// Busca tempo de ciclo instantâneo/corrente das tarefas
GetTaskInfo (psAppName, Task_Information.TI_MainTask.psTaskName, Task_Information.TI_MainTask.pstTaskInfo);
GetTaskInfo (psAppName, Task_Information.TI_Configuration.psTaskName, Task_Information.TI_Configuration.pstTaskInfo);
GetTaskInfo (psAppName, Task_Information.TI_MODBUS_Client_2.psTaskName, Task_Information.TI_MODBUS_Client_2.pstTaskInfo);
GetTaskInfo (psAppName, Task_Information.TI_MODBUS_Client_3.psTaskName, Task_Information.TI_MODBUS_Client_3.pstTaskInfo);
GetTaskInfo (psAppName, Task_Information.TI_MODBUS_Master_1.psTaskName, Task_Information.TI_MODBUS_Master_1.pstTaskInfo);
GetTaskInfo (psAppName, Task_Information.TI_MODBUS_Server_2.psTaskName, Task_Information.TI_MODBUS_Server_2.pstTaskInfo);
GetTaskInfo (psAppName, Task_Information.TI_MODBUS_Server_3.psTaskName, Task_Information.TI_MODBUS_Server_3.pstTaskInfo);
GetTaskInfo (psAppName, Task_Information.TI_MODBUS_Slave_1.psTaskName, Task_Information.TI_MODBUS_Slave_1.pstTaskInfo);


// Se este for o PLCA e ele está no estado ativo...
IF DG_NX4010.tRedundancy.RedDgnLoc.sGeneral_Diag.ePLC_ID = CLUCONF_ID.PLC_A AND
   DG_NX4010.tRedundancy.RedDgnLoc.sGeneral_Diag.eRedState = REDUNDANCY_STATE.ACTIVE THEN
   
   	// Indica que existe um PLC ativo
	bPouActiveTime:= TRUE;
	
	// Atualiza variáveis de tempo de ciclo instantâneo/corrente das tarefas
	PersistentVars.dwPLCAMainTaskCurScanTime:= Task_Information.TI_MainTask.TaskInfo.dwCurScanTime;
	PersistentVars.dwPLCAConfigurationCurScanTime:= Task_Information.TI_Configuration.TaskInfo.dwCurScanTime;

	// Reseta variáveis de tempo de ciclo máximo e mínimo das tarefas caso solicitado
	IF Symbolics.bPlcAMaxMinSetup = TRUE THEN
		Symbolics.bPlcAMaxMinSetup:= FALSE;
		PersistentVars.dwPLCAMainTaskMaxScanTime:= PersistentVars.dwPLCAMainTaskCurScanTime;
		PersistentVars.dwPLCAMainTaskMinScanTime:= PersistentVars.dwPLCAMainTaskCurScanTime;
		PersistentVars.dwPLCAConfigurationMaxScanTime:= PersistentVars.dwPLCAConfigurationCurScanTime;
		PersistentVars.dwPLCAConfigurationMinScanTime:= PersistentVars.dwPLCAConfigurationCurScanTime;
	END_IF
	
	// Atualiza variáveis de tempo de ciclo máximo e mínimo das tarefas
	PersistentVars.dwPLCAMainTaskMaxScanTime:= MAX(PersistentVars.dwPLCAMainTaskMaxScanTime, PersistentVars.dwPLCAMainTaskCurScanTime);
	PersistentVars.dwPLCAMainTaskMinScanTime:= MIN(PersistentVars.dwPLCAMainTaskMinScanTime, PersistentVars.dwPLCAMainTaskCurScanTime);
	PersistentVars.dwPLCAConfigurationMaxScanTime:= MAX(PersistentVars.dwPLCAConfigurationMaxScanTime, PersistentVars.dwPLCAConfigurationCurScanTime);
	PersistentVars.dwPLCAConfigurationMinScanTime:= MIN(PersistentVars.dwPLCAConfigurationMinScanTime, PersistentVars.dwPLCAConfigurationCurScanTime);
	
	// Calcula tempo de ciclo médio da tarefa principal
	dwMainTaskSum:= dwMainTaskSum - adwAvgMainTask[iMainIndex];
	adwAvgMainTask[iMainIndex]:= PersistentVars.dwPLCAMainTaskCurScanTime;
	dwMainTaskSum:= dwMainTaskSum + adwAvgMainTask[iMainIndex];
	iMainIndex:= iMainIndex + 1;
	IF iMainIndex > DWORD_TO_INT(SIZEOF(adwAvgMainTask)/SIZEOF(adwAvgMainTask[1])) THEN
		iMainIndex:= 1;
	END_IF
	
	// Calcula tempo de ciclo médio da tarefa de configuração
	dwConfigTaskSum:= dwConfigTaskSum - adwAvgConfigTask[iConfigIndex];
	adwAvgConfigTask[iConfigIndex]:= PersistentVars.dwPLCAConfigurationCurScanTime;
	dwConfigTaskSum:= dwConfigTaskSum + adwAvgConfigTask[iConfigIndex];
	iConfigIndex:= iConfigIndex + 1;
	IF iConfigIndex > DWORD_TO_INT(SIZEOF(adwAvgConfigTask)/SIZEOF(adwAvgConfigTask[1])) THEN
		iConfigIndex:= 1;
	END_IF
	
	// Atualiza variáveis de tempo de ciclo médio das tarefas
	PersistentVars.dwPLCAMainTaskAvgScanTime:= dwMainTaskSum/(SIZEOF(adwAvgMainTask)/SIZEOF(adwAvgMainTask[1]));
	PersistentVars.dwPLCAConfigurationAvgScanTime:= dwConfigTaskSum/(SIZEOF(adwAvgConfigTask)/SIZEOF(adwAvgConfigTask[1]));

	// Registra percentual de uso da MainTask
	PersistentVars.dwPLCAMainTaskLoadMax:= MAX(PersistentVars.dwPLCAMainTaskLoadMax, (PersistentVars.dwPLCAMainTaskCurScanTime)/INT_TO_DWORD(ProjectConstants.iMainTaskInterval));
	PersistentVars.dwPLCAMainTaskLoadAvg:= (PersistentVars.dwPLCAMainTaskAvgScanTime)/INT_TO_DWORD(ProjectConstants.iMainTaskInterval);
	PersistentVars.dwPLCAMainTaskLoadMin:= MIN(PersistentVars.dwPLCAMainTaskLoadMin, (PersistentVars.dwPLCAMainTaskCurScanTime)/INT_TO_DWORD(ProjectConstants.iMainTaskInterval));
END_IF

// Se este for o PLCB e ele está no estado ativo...
IF DG_NX4010.tRedundancy.RedDgnLoc.sGeneral_Diag.ePLC_ID = CLUCONF_ID.PLC_B AND
   DG_NX4010.tRedundancy.RedDgnLoc.sGeneral_Diag.eRedState = REDUNDANCY_STATE.ACTIVE THEN
	
   	// Indica que existe um PLC ativo
	bPouActiveTime:= TRUE;
	
	// Atualiza variáveis de tempo de ciclo instantâneo/corrente das tarefas
	PersistentVars.dwPLCBMainTaskCurScanTime:= Task_Information.TI_MainTask.TaskInfo.dwCurScanTime;
	PersistentVars.dwPLCBConfigurationCurScanTime:= Task_Information.TI_Configuration.TaskInfo.dwCurScanTime;
	
	// Reseta variáveis de tempo de ciclo máximo e mínimo das tarefas caso solicitado
	IF Symbolics.bPlcBMaxMinSetup = TRUE THEN
		Symbolics.bPlcBMaxMinSetup:= FALSE;	
		PersistentVars.dwPLCBMainTaskMaxScanTime:= PersistentVars.dwPLCBMainTaskCurScanTime;
		PersistentVars.dwPLCBMainTaskMinScanTime:= PersistentVars.dwPLCBMainTaskCurScanTime;
		PersistentVars.dwPLCBConfigurationMaxScanTime:= PersistentVars.dwPLCBConfigurationCurScanTime;
		PersistentVars.dwPLCBConfigurationMinScanTime:= PersistentVars.dwPLCBConfigurationCurScanTime;
	END_IF
	
	// Atualiza variáveis de tempo de ciclo máximo e mínimo das tarefas
	PersistentVars.dwPLCBMainTaskMaxScanTime:= MAX(PersistentVars.dwPLCBMainTaskMaxScanTime, PersistentVars.dwPLCBMainTaskCurScanTime);
	PersistentVars.dwPLCBMainTaskMinScanTime:= MIN(PersistentVars.dwPLCBMainTaskMinScanTime, PersistentVars.dwPLCBMainTaskCurScanTime);
	PersistentVars.dwPLCBConfigurationMaxScanTime:= MAX(PersistentVars.dwPLCBConfigurationMaxScanTime, PersistentVars.dwPLCBConfigurationCurScanTime);
	PersistentVars.dwPLCBConfigurationMinScanTime:= MIN(PersistentVars.dwPLCBConfigurationMinScanTime, PersistentVars.dwPLCBConfigurationCurScanTime);
	
	// Calcula tempo de ciclo médio da tarefa principal
	dwMainTaskSum:= dwMainTaskSum - adwAvgMainTask[iMainIndex];
	adwAvgMainTask[iMainIndex]:= PersistentVars.dwPLCBMainTaskCurScanTime;
	dwMainTaskSum:= dwMainTaskSum + adwAvgMainTask[iMainIndex];
	iMainIndex:= iMainIndex + 1;
	IF iMainIndex > DWORD_TO_INT(SIZEOF(adwAvgMainTask)/SIZEOF(adwAvgMainTask[1])) THEN
		iMainIndex:= 1;
	END_IF
	
	// Calcula tempo de ciclo médio da tarefa de configuração
	dwConfigTaskSum:= dwConfigTaskSum - adwAvgConfigTask[iConfigIndex];
	adwAvgConfigTask[iConfigIndex]:= PersistentVars.dwPLCBConfigurationCurScanTime;
	dwConfigTaskSum:= dwConfigTaskSum + adwAvgConfigTask[iConfigIndex];
	iConfigIndex:= iConfigIndex + 1;
	IF iConfigIndex > DWORD_TO_INT(SIZEOF(adwAvgConfigTask)/SIZEOF(adwAvgConfigTask[1])) THEN
		iConfigIndex:= 1;
	END_IF
	
	// Atualiza variáveis de tempo de ciclo médio das tarefas
	PersistentVars.dwPLCBMainTaskAvgScanTime:= dwMainTaskSum/(SIZEOF(adwAvgMainTask)/SIZEOF(adwAvgMainTask[1]));
	PersistentVars.dwPLCBConfigurationAvgScanTime:= dwConfigTaskSum/(SIZEOF(adwAvgConfigTask)/SIZEOF(adwAvgConfigTask[1]));
	
	// Registra percentual de uso da MainTask
	PersistentVars.dwPLCBMainTaskLoadMax:= MAX(PersistentVars.dwPLCBMainTaskLoadMax, (PersistentVars.dwPLCBMainTaskCurScanTime)/INT_TO_DWORD(ProjectConstants.iMainTaskInterval));
	PersistentVars.dwPLCBMainTaskLoadAvg:= (PersistentVars.dwPLCBMainTaskAvgScanTime)/INT_TO_DWORD(ProjectConstants.iMainTaskInterval);
	PersistentVars.dwPLCBMainTaskLoadMin:= MIN(PersistentVars.dwPLCBMainTaskLoadMin, (PersistentVars.dwPLCBMainTaskCurScanTime)/INT_TO_DWORD(ProjectConstants.iMainTaskInterval));
END_IF

// Calcula o tempo mínimo total, somando a duração mínima de todas as POUs, menos da MainPrg
MinMaxTimes.uliPouMinTime_TOTAL:=	MinMaxTimes.uliPouMinTime_Alarms +
						MinMaxTimes.uliPouMinTime_CheckIec104 +
						MinMaxTimes.uliPouMinTime_CheckLanguages +
						MinMaxTimes.uliPouMinTime_CheckProfibusIOs +
						MinMaxTimes.uliPouMinTime_CheckRecipe +
						MinMaxTimes.uliPouMinTime_CheckSoe +
						MinMaxTimes.uliPouMinTime_IncrRedData +
						MinMaxTimes.uliPouMinTime_PidGenerator +
						MinMaxTimes.uliPouMinTime_StateChange +
						MinMaxTimes.uliPouMinTime_CheckDiags +
						MinMaxTimes.uliPouMinTime_CheckForcing +		
						MinMaxTimes.uliPouMinTime_CheckModbus1 +
						MinMaxTimes.uliPouMinTime_CheckModbus2 +
						MinMaxTimes.uliPouMinTime_CheckModbus3 +
						MinMaxTimes.uliPouMinTime_CheckModbus4 +
						MinMaxTimes.uliPouMinTime_CheckRam +
						MinMaxTimes.uliPouMinTime_CheckRedData +
						MinMaxTimes.uliPouMinTime_CheckSntp +
						MinMaxTimes.uliPouMinTime_CleanStatus +
						MinMaxTimes.uliPouMinTime_CycleTimes +
						//MinMaxTimes.uliPouMinTime_DaylightSavingTime +
						MinMaxTimes.uliPouMinTime_UserLog +
						MinMaxTimes.uliPouMinTime_WriteHwVersionsNonActive+
						MinMaxTimes.uliPouMinTime_CheckNVL +
						MinMaxTimes.uliPouMinTime_MQTT;
						
// Calcula o tempo máximo total, somando a duração máxima de todas as POUs, menos da MainPrg
MinMaxTimes.uliPouMaxTime_TOTAL:=	MinMaxTimes.uliPouMaxTime_Alarms +
						MinMaxTimes.uliPouMaxTime_CheckIec104 +
						MinMaxTimes.uliPouMaxTime_CheckLanguages +
						MinMaxTimes.uliPouMaxTime_CheckProfibusIOs + 
						MinMaxTimes.uliPouMaxTime_CheckRecipe +
						MinMaxTimes.uliPouMaxTime_CheckSoe +
						MinMaxTimes.uliPouMaxTime_IncrRedData +
						MinMaxTimes.uliPouMaxTime_PidGenerator +
						MinMaxTimes.uliPouMaxTime_StateChange +
						MinMaxTimes.uliPouMaxTime_CheckDiags +
						MinMaxTimes.uliPouMaxTime_CheckForcing +		
						MinMaxTimes.uliPouMaxTime_CheckModbus1 +
						MinMaxTimes.uliPouMaxTime_CheckModbus2 +
						MinMaxTimes.uliPouMaxTime_CheckModbus3 +
						MinMaxTimes.uliPouMaxTime_CheckModbus4 +
						MinMaxTimes.uliPouMaxTime_CheckRam +
						MinMaxTimes.uliPouMaxTime_CheckRedData +
						MinMaxTimes.uliPouMaxTime_CheckSntp +
						MinMaxTimes.uliPouMaxTime_CleanStatus +
						MinMaxTimes.uliPouMaxTime_CycleTimes +
						//MinMaxTimes.uliPouMaxTime_DaylightSavingTime +
						MinMaxTimes.uliPouMaxTime_UserLog +
						MinMaxTimes.uliPouMaxTime_WriteHwVersionsNonActive+
						MinMaxTimes.uliPouMaxTime_CheckNVL+
						MinMaxTimes.uliPouMaxTime_MQTT;

// Registra o tempo do sistema
SysTimeGetUs(uliPouEndTime);
// Calcula duração mínima/máxima desta POU, se um dos PLCs está ativo
IF bPouActiveTime THEN
	MinMaxTimes.uliPouMinTime_CycleTimes:= MIN(MinMaxTimes.uliPouMinTime_CycleTimes, uliPouEndTime - uliPouIniTime);
	MinMaxTimes.uliPouMaxTime_CycleTimes:= MAX(MinMaxTimes.uliPouMaxTime_CycleTimes, uliPouEndTime - uliPouIniTime);
END_IF

END_PROGRAM

// Device/Application/UserPOUs/Non-Redundant/CheckModbus1
PROGRAM CheckModbus1
VAR
	byIndex : BYTE;
	wIndex : WORD;
	bStatusCoil : BOOL;
	bStatusStatus : BOOL;
	bStatusHolding : BOOL;
	bStatusInputReg : BOOL;
	liDigitalTimer : LINT := 0;
	liAnalogTimer : LINT := 0;
	abyCoilsError_DataWr : ARRAY [0..119] OF BYTE;
	abyCoilsError_DataRd : ARRAY [0..119] OF BYTE;
	abyStatusError_DataWr : ARRAY [0..119] OF BYTE;
	abyStatusError_DataRd : ARRAY [0..119] OF BYTE;
	awHoldingError_DataWr : ARRAY [0..119] OF WORD;
	awHoldingError_DataRd : ARRAY [0..119] OF WORD;
	awInputRegError_DataWr : ARRAY [0..119] OF WORD;
	awInputRegError_DataRd : ARRAY [0..119] OF WORD;
	wOldRXNormalResponses : WORD;
	iMilisecondsCounter : INT;
	iBytesPerResponse : INT := 240;
	uliPouIniTime : ULINT;
	uliPouEndTime : ULINT;
END_VAR

// Consistencia da integridade dos dados trocados via MODBUS 1

// Registra o tempo do sistema
SysTimeGetUs(uliPouIniTime);

//
// Controle e consistência dos coils e input status
//

// Consiste os valores lidos
bStatusCoil:= TRUE;
bStatusStatus:= TRUE;
FOR byIndex:= 0 TO 119 BY 1 DO
	bStatusCoil:= bStatusCoil AND (ATs.abyModbus1CoilsRead[byIndex] = ATs.abyModbus1CoilsWrite[byIndex]);
	bStatusStatus:= bStatusStatus AND (ATs.abyModbus1StatusRead[byIndex] = ATs.abyModbus1CoilsWrite[byIndex]);
END_FOR

// Se o protocolo MODBUS está rodando e se os dados são consistentes...
IF DG_MODBUS_Master_1.tDiag.bRunning AND bStatusCoil AND bStatusStatus THEN
	// Altera o valor a ser escrito nos coils
	ATs.abyModbus1CoilsWrite[0]:= ATs.abyModbus1CoilsWrite[0] + 10;
	// Reseta o temporizador
	liDigitalTimer:= 0;
ELSE
	// Acumula o tempo que passou
	liDigitalTimer:= liDigitalTimer + ProjectConstants.iMainTaskInterval;
	// Registra o tempo máximo
	MinMaxTimes.liDigMaxTime_CheckModbus1:= MAX(MinMaxTimes.liDigMaxTime_CheckModbus1, liDigitalTimer);
	// Caso o tempo máximo tenha sido extrapolado...
	IF liDigitalTimer >= ProjectConstants.iModbus1ReadWriteDelay THEN
		// Registra falha nos coils, caso tenha ocorrido
		IF bStatusCoil = FALSE THEN
			NonRedPointer.pbModbus1ErrorCoilLoc^:= TRUE;
			abyCoilsError_DataWr:= ATs.abyModbus1CoilsWrite;
			abyCoilsError_DataRd:= ATs.abyModbus1CoilsRead;		
		END_IF
		// Registra falha nos inputs, caso tenha ocorrido
		IF bStatusStatus = FALSE THEN
			NonRedPointer.pbModbus1ErrorStatusLoc^:= TRUE;
			abyStatusError_DataWr:= ATs.abyModbus1CoilsWrite;
			abyStatusError_DataRd:= ATs.abyModbus1StatusRead;
		END_IF
	END_IF
END_IF

// Atualiza os valores escritos
FOR byIndex:= 1 TO 119 BY 1 DO
	ATs.abyModbus1CoilsWrite[byIndex]:= ATs.abyModbus1CoilsWrite[byIndex - 1] + byIndex;
END_FOR

//
// Controle e consistência dos holding e input registers
//

// Consiste os valores lidos
bStatusHolding:= TRUE;
bStatusInputReg:= TRUE;
FOR wIndex:= 0 TO 119 BY 1 DO
	bStatusHolding:= bStatusHolding AND (ATs.awModbus1HoldingRead[wIndex] = ATs.awModbus1HoldingWrite[wIndex]);
	bStatusInputReg:= bStatusInputReg AND (ATs.awModbus1InputRegRead[wIndex] = ATs.awModbus1HoldingWrite[wIndex]);
END_FOR

// Se o protocolo MODBUS está rodando e se os dados são consistentes...
IF DG_MODBUS_Master_1.tDiag.bRunning AND bStatusHolding AND bStatusInputReg THEN
	// Incrementa o valor escrito nos holding registers
	ATs.awModbus1HoldingWrite[0]:= ATs.awModbus1HoldingWrite[0] + 100;
	// Reseta o temporizador
	liAnalogTimer:= 0;
ELSE
	// Acumula o tempo que passou
	liAnalogTimer:= liAnalogTimer + ProjectConstants.iMainTaskInterval;
	// Registra o tempo máximo
	MinMaxTimes.liAnaMaxTime_CheckModbus1:= MAX(MinMaxTimes.liAnaMaxTime_CheckModbus1, liAnalogTimer);
	// Caso o tempo máximo tenha sido extrapolado...
	IF liAnalogTimer >= ProjectConstants.iModbus1ReadWriteDelay THEN
		// Registra falha nos holding register, caso tenha ocorrido
		IF bStatusHolding = FALSE THEN
			NonRedPointer.pbModbus1ErrorHoldingLoc^:= TRUE;
			awHoldingError_DataWr:= ATs.awModbus1HoldingWrite;
			awHoldingError_DataRd:= ATs.awModbus1HoldingRead;
		END_IF
		// Registra falha nos input register, caso tenha ocorrido
		IF bStatusInputReg = FALSE THEN
			NonRedPointer.pbModbus1ErrorInputRegLoc^:= TRUE;
			awInputRegError_DataWr:= ATs.awModbus1HoldingWrite;
			awInputRegError_DataRd:= ATs.awModbus1InputRegRead;
		END_IF
	END_IF
END_IF

// Atualiza os valores escritos
FOR wIndex:= 1 TO 119 BY 1 DO
	ATs.awModbus1HoldingWrite[wIndex]:= ATs.awModbus1HoldingWrite[wIndex - 1] + wIndex;
END_FOR

//
// Calcula a taxa média de comunicação
//

// Incrementa o número de milisegundos que transcorreram
iMilisecondsCounter:= iMilisecondsCounter + ProjectConstants.iMainTaskInterval;
// Se já se passou o tempo configurado desde a última média realizada...
IF iMilisecondsCounter >= ProjectConstants.iMsToComputeComRate THEN
	// Só calcula se o contador não virou
	IF DG_MODBUS_Master_1.tStat.wRXNormalResponses > wOldRXNormalResponses THEN
		// Calcula a taxa de comunicação atual
		MinMaxTimes.diModbus1BytesPerSec:=	WORD_TO_DINT(DG_MODBUS_Master_1.tStat.wRXNormalResponses - wOldRXNormalResponses) *
											iBytesPerResponse * 1000 / iMilisecondsCounter;
	END_IF
	// Zera o número de milisegundos transcorridos
	iMilisecondsCounter:= 0;
	// Salva número de respostas atuais
	wOldRXNormalResponses:= DG_MODBUS_Master_1.tStat.wRXNormalResponses;
END_IF

PersistentVars.bModbus1ErrorCoil:=		NonRedPointer.pbModbus1ErrorCoilLoc^ OR
										NonRedPointer.pbModbus1ErrorCoilRem^;
PersistentVars.bModbus1ErrorStatus:=	NonRedPointer.pbModbus1ErrorStatusLoc^ OR
										NonRedPointer.pbModbus1ErrorStatusRem^;
PersistentVars.bModbus1ErrorHolding:=	NonRedPointer.pbModbus1ErrorHoldingLoc^ OR
										NonRedPointer.pbModbus1ErrorHoldingRem^;
PersistentVars.bModbus1ErrorInputReg:=	NonRedPointer.pbModbus1ErrorInputRegLoc^ OR
										NonRedPointer.pbModbus1ErrorInputRegRem^;

// Registra o tempo do sistema
SysTimeGetUs(uliPouEndTime);
// Calcula duração mínima/máxima desta POU
MinMaxTimes.uliPouMinTime_CheckModbus1:= MIN(MinMaxTimes.uliPouMinTime_CheckModbus1, uliPouEndTime - uliPouIniTime);
MinMaxTimes.uliPouMaxTime_CheckModbus1:= MAX(MinMaxTimes.uliPouMaxTime_CheckModbus1, uliPouEndTime - uliPouIniTime);

END_PROGRAM

// Device/Application/UserPOUs/Redundant/ProfibusStateChange
PROGRAM ProfibusStateChange
VAR
	byState : BYTE := 1;
	iTime : INT := 0;
	iLimit : INT := ProjectConstants.iLowLimit;
	bLastState : BOOL;
	uliPouIniTime : ULINT;
	uliPouEndTime : ULINT;
END_VAR

 // Esta POU alterna o estado de redundância das remotas Profibus automaticamente.
// Ela é chamada pela POU CheckProfibusIOs, portanto ela é executada somente pelo CP ativo,
// isto deve ser levado em consideração para compreender o código abaixo.
// Estado inicial: Remota A ativo, Remota B stand-by.

// Registra o tempo do sistema
SysTimeGetUs(uliPouIniTime);

CASE byState OF
	
	1:	// Aguarda tempo para estabilização da nova remota ativa
		IF iTime < ProjectConstants.iTimeToSkipAsActive THEN
			iTime:= iTime + ProjectConstants.iMainTaskInterval;
		ELSE
			// Próximo estado
			byState:= 2;
			// Joga zero para os bits de switch over das remotas ponto para que estas o executem
			REM05_PO5065_OUT:= 0;
			REM10_PO5065_OUT:= 0;
		END_IF
	
	2:	// Aguarda iLimit ciclos para a próxima alteração de estados
		IF iTime < iLimit THEN
			iTime:= iTime + ProjectConstants.iMainTaskInterval;
		ELSE
			byState:= 3;
		END_IF
	
	3:	// Realiza switchover
		PersistentVars.dwPBSwitchoverCnt:= PersistentVars.dwPBSwitchoverCnt + 1;
		IF bLastState THEN
			REM05_PO5065_OUT:= 1024;
			REM10_PO5065_OUT:= 1024;
			bLastState:=FALSE;
		ELSE
			REM05_PO5065_OUT:= 768;
			REM10_PO5065_OUT:= 768;
			bLastState:=TRUE;
		END_IF			
		byState:= 4;
		iTime:= 0;
			
	4: 	// Incrementa o valor limite para troca de estados
		iLimit:= iLimit + ProjectConstants.iMainTaskInterval;
		// Mantém a duração de cada estado entre 50 e 250 ciclos
		IF iLimit > ProjectConstants.iHighLimit THEN
			iLimit:= ProjectConstants.iLowLimit;
		END_IF
		// Inicia um novo ciclo de troca de estados
		byState:= 1;
END_CASE

// Registra o tempo do sistema
SysTimeGetUs(uliPouEndTime);
// Calcula duração mínima/máxima desta POU
MinMaxTimes.uliPouMinTime_ProfibusStateChange:= MIN(MinMaxTimes.uliPouMinTime_ProfibusStateChange, uliPouEndTime - uliPouIniTime);
MinMaxTimes.uliPouMaxTime_ProfibusStateChange:= MAX(MinMaxTimes.uliPouMaxTime_ProfibusStateChange, uliPouEndTime - uliPouIniTime);

END_PROGRAM

// Device/Application/UserPOUs/Non-Redundant/CheckRam
PROGRAM CheckRam
VAR
	stRamInfo : SYSTEM_RAM_INFO_T;
	dwRamTotalError : DWORD;
	dwRamFreeError : DWORD;
	uliPouIniTime : ULINT;
	uliPouEndTime : ULINT;
	bInternalFlag : BOOL;
END_VAR

// POU para consistência da memória RAM total e livre.

// Registra o tempo do sistema
SysTimeGetUs(uliPouIniTime);

// Busca as informações da memória RAM apenas no primeiro ciclo como inativo, pois a função consome muito tempo
IF DG_NX4010.tRedundancy.RedDgnLoc.sGeneral_Diag.eRedState = REDUNDANCY_STATE.INACTIVE  AND NonRedData.bRedStateChanged  THEN
	// Atualiza as informações a respeito da memória RAM
	SystemRamInfoGet(stRamInfo);
	// Flag para indicar se passou pelo estado inativo para habiltiar a consistencia do teste na inicialização do teste
	IF stRamInfo.dwTotal > 0 AND stRamInfo.dwFree > 0 THEN
		bInternalFlag:= TRUE;
	END_IF
END_IF

// Consiste a memória RAM apenas no primeiro ciclo como ativo (a UCP não ativa não consegue escrever nas PersistentVars)  
IF 	DG_NX4010.tRedundancy.RedDgnLoc.sGeneral_Diag.eRedState = REDUNDANCY_STATE.ACTIVE AND NonRedData.bRedStateChanged AND bInternalFlag THEN

		// Consistência da memória RAM total
		IF stRamInfo.dwTotal <> ProjectConstants.dwRamTotal THEN
			dwRamTotalError:= stRamInfo.dwTotal;
			NonRedPointer.pbRamTotalFailureLoc^:= TRUE;
		END_IF
	// Registra os valores mínimos e máximos e consiste a variação de memória livre
			IF DG_NX4010.tRedundancy.RedDgnLoc.sGeneral_Diag.ePLC_ID = CLUCONF_ID.PLC_A THEN
				// Registra valores de memória RAM livre mínima e máxima do PLC correspondente
				PersistentVars.dwMinFreeRamPlcA:= MIN(PersistentVars.dwMinFreeRamPlcA, stRamInfo.dwFree/1024);
				PersistentVars.dwMaxFreeRamPlcA:= MAX(PersistentVars.dwMaxFreeRamPlcA, stRamInfo.dwFree/1024);
				PersistentVars.dwInstFreeRamPlcA:= stRamInfo.dwFree/1024;
				// Consistência da variação da memória RAM livre
				IF PersistentVars.dwMaxFreeRamPlcA - PersistentVars.dwMinFreeRamPlcA > ProjectConstants.dwRamVariance THEN
					dwRamFreeError:= PersistentVars.dwMaxFreeRamPlcA;
					NonRedPointer.pbRamFreeVarFailureLoc^:= TRUE;
				END_IF
			ELSE
				// Registra valores de memória RAM livre mínima e máxima do PLC correspondente
				PersistentVars.dwMinFreeRamPlcB:= MIN(PersistentVars.dwMinFreeRamPlcB, stRamInfo.dwFree/1024);
				PersistentVars.dwMaxFreeRamPlcB:= MAX(PersistentVars.dwMaxFreeRamPlcB, stRamInfo.dwFree/1024);
				PersistentVars.dwInstFreeRamPlcB:= stRamInfo.dwFree/1024;
				// Consistência da variação da memória RAM livre
				IF PersistentVars.dwMaxFreeRamPlcB - PersistentVars.dwMinFreeRamPlcB > ProjectConstants.dwRamVariance THEN
					dwRamFreeError:= PersistentVars.dwMaxFreeRamPlcB;
					NonRedPointer.pbRamFreeVarFailureLoc^:= TRUE;
				END_IF
			END_IF
	// Reinicializa flag de teste
	bInternalFlag:= FALSE;
END_IF

// Inicializa os diagnósticos locais/remotos se solicitado
IF SymbolicsNonRedundant.bEnableCleanStats_CheckRam THEN
	NonRedPointer.pbRamTotalFailureLoc^:= FALSE;
	NonRedPointer.pbRamFreeVarFailureLoc^:= FALSE;
	NonRedPointer.pbRamTotalFailureRem^:= FALSE;
	NonRedPointer.pbRamFreeVarFailureRem^:= FALSE;	
	// Reinicializa flag de teste
	bInternalFlag:= FALSE;
	// Inicializa os valores atualizados pela função SystemRamInfoGet
	stRamInfo.dwTotal:= 0;
	stRamInfo.dwFree:= 0;
	SymbolicsNonRedundant.bEnableCleanStats_CheckRam := FALSE;
END_IF

// Atribui as variáveis locais/remotas de falha às variáveis redundantes persistentes

PersistentVars.bRamTotalFailure:=	PersistentVars.bRamTotalFailure OR
									NonRedPointer.pbRamTotalFailureLoc^ OR
									NonRedPointer.pbRamTotalFailureRem^;
PersistentVars.bRamFreeVarFailure:=	PersistentVars.bRamFreeVarFailure OR
									NonRedPointer.pbRamFreeVarFailureLoc^ OR
									NonRedPointer.pbRamFreeVarFailureRem^;

// Registra o tempo do sistema
SysTimeGetUs(uliPouEndTime);
// Calcula duração mínima/máxima desta POU
MinMaxTimes.uliPouMinTime_CheckRam:= MIN(MinMaxTimes.uliPouMinTime_CheckRam, uliPouEndTime - uliPouIniTime);
MinMaxTimes.uliPouMaxTime_CheckRam:= MAX(MinMaxTimes.uliPouMaxTime_CheckRam, uliPouEndTime - uliPouIniTime);

END_PROGRAM

// Device/Application/UserPOUs/Non-Redundant/CheckSntp
PROGRAM CheckSntp
VAR CONSTANT
	byDelay : BYTE := 10;
	iSntpTolerance : INT := (21200); // = 20000 + 1200
END_VAR
VAR
	sCurrentTime : NextoStandard.EXTENDED_DATE_AND_TIME;
	sGetTime : NextoStandard.EXTENDED_DATE_AND_TIME;
	sSetTime : NextoStandard.SetDateAndTime;
	GetTimeZone_Status : RTC_STATUS;
	TimeZone : TIMEZONESETTINGS;
	bStartup : BOOL := TRUE;
	byState : BYTE := 1;
	bSignal : BOOL := FALSE;
	iSyncCounter : INT := 0;
	dwReference : DWORD := 0;
	liSntpMsTimer : LINT := 0;
	uliPouIniTime : ULINT;
	uliPouEndTime : ULINT;
END_VAR

// Teste que verifica a atualização do relógio pelo SNTP
// SETUP: Configurar o SNTP para 20s de period, com 150ms de minimum error

// Registra o tempo do sistema
SysTimeGetUs(uliPouIniTime);

// Testa se a função GetTimeZone estrá retornando os valores corretos
GetTimeZone_Status := GetTimeZone(TimeZone);
IF GetTimeZone_Status <> RTC_STATUS.NO_ERROR OR TimeZone.iHour <> -3 OR TimeZone.iMinutes <> 0 THEN
	PersistentVars.bTimezoneFailure := TRUE;
END_IF

// Acumula o tempo que passou
liSntpMsTimer:= liSntpMsTimer + ProjectConstants.iMainTaskInterval;

// Verifica se o serviço está funcionando
IF	DG_NX3030.tDetailed.SNTP.bServiceEnabled = TRUE AND
	DG_NX3030.tDetailed.SNTP.byActiveTimeServer <> NO_TIME_SERVER THEN
		// Correção inicial da referência
		IF bStartup = TRUE THEN
			// Correção inicial da referência
			dwReference:= DG_NX3030.tDetailed.SNTP.dwRTCTimeUpdatedCount;
			// Restaura variáveis locais não retentivas
			NonRedPointer.pbSntpServerFailuresLoc^:= PersistentVars.bSntpServerFailures;
			NonRedPointer.pbSntpSourceFailuresLoc^:= PersistentVars.bSntpSourceFailures;
			NonRedPointer.piSntpSyncFailuresLoc^:= PersistentVars.iSntpSyncFailures;
			// Reseta indicação de inicialização
			bStartup:= FALSE;
		END_IF
		
		CASE byState OF
			
			1:	// Armazena o horário atual em sCurrentTime, confere se a atualização anterior ocorreu
				NextoStandard.GetDateAndTime(sGetTime);
				sCurrentTime.byDayOfMonth:= sGetTime.byDayOfMonth;
				sCurrentTime.byHours:= sGetTime.byHours;
				sCurrentTime.byMinutes:= sGetTime.byMinutes;
				sCurrentTime.byMonth:= sGetTime.byMonth;
				sCurrentTime.bySeconds:= sGetTime.bySeconds;
				sCurrentTime.wMilliseconds:= sGetTime.wMilliseconds;
				sCurrentTime.wYear:= sGetTime.wYear;
				// Se o contador está diferente da referência, indica erro na sincronização
				IF DG_NX3030.tDetailed.SNTP.dwRTCTimeUpdatedCount < dwReference THEN
					IF NonRedPointer.piSntpSyncFailuresLoc^ < ProjectConstants.iValueRedLimit THEN
						NonRedPointer.piSntpSyncFailuresLoc^:= NonRedPointer.piSntpSyncFailuresLoc^+1;
					END_IF
					dwReference:= DG_NX3030.tDetailed.SNTP.dwRTCTimeUpdatedCount;
				// Indica que houve 2 atualizações no intervalo, o que não pode ser considerado uma falha
				ELSIF DG_NX3030.tDetailed.SNTP.dwRTCTimeUpdatedCount > dwReference THEN
					dwReference:= DG_NX3030.tDetailed.SNTP.dwRTCTimeUpdatedCount;
				END_IF				
				byState:= 2;
			
			2:	// Adianta ou atrasa sCurrentTime em 10s alternadamente
				IF bSignal = TRUE THEN
					IF sCurrentTime.bySeconds >= byDelay THEN
						sCurrentTime.bySeconds:= sCurrentTime.bySeconds - byDelay;
						byState:= 3;
					ELSE
						byState:= 1;
					END_IF
				ELSE
					IF sCurrentTime.bySeconds < (60 - byDelay) THEN
						sCurrentTime.bySeconds:= sCurrentTime.bySeconds + byDelay;
						byState:= 3;
					ELSE
						byState:= 1;
					END_IF
				END_IF
			
			3:	// Aplica o horário com 10s de erro ao relógio
				bSignal:= NOT(bSignal);
				sSetTime.DATEANDTIME.byDayOfMonth:= sCurrentTime.byDayOfMonth;
				sSetTime.DATEANDTIME.byHours:= sCurrentTime.byHours;
				sSetTime.DATEANDTIME.byMinutes:= sCurrentTime.byMinutes;
				sSetTime.DATEANDTIME.byMonth:= sCurrentTime.byMonth;
				sSetTime.DATEANDTIME.bySeconds:= sCurrentTime.bySeconds;
				sSetTime.DATEANDTIME.wMilliseconds:= sCurrentTime.wMilliseconds;
				sSetTime.DATEANDTIME.wYear:= sCurrentTime.wYear;
				sSetTime(REQUEST:= TRUE);
				IF sSetTime.DONE = TRUE THEN
					sSetTime(REQUEST:= FALSE);
					byState:= 4;
				END_IF
			
			4:	// Aguarda 20s, que é o período de sincronização, + tolerância de 1,2s
				iSyncCounter:= iSyncCounter + 1;
				IF iSyncCounter = (iSntpTolerance/ProjectConstants.iMainTaskInterval) THEN
					iSyncCounter:= 0;
					byState:= 5;
				END_IF
			
			5:	// Aguarda passagem do tempo configurado para o próximo teste
				IF liSntpMsTimer >= ProjectConstants.liClockSyncDelay THEN
					dwReference:= dwReference + 1;
					liSntpMsTimer:= 0;
					byState:= 1;
				END_IF			
		END_CASE
ELSE
	// Desconsidera as falhas até 15 segundos após a inicialização do sistema
	IF bStartup = FALSE OR liSntpMsTimer > 15000 THEN
		// Incrementa contador de falhas por falta de fonte de sincronismo
		IF DG_NX3030.tDetailed.SNTP.bServiceEnabled = FALSE THEN
			NonRedPointer.pbSntpSourceFailuresLoc^:= TRUE;
		END_IF
		// Incrementa falha por falta de servidor SNTP
		IF DG_NX3030.tDetailed.SNTP.byActiveTimeServer = NO_TIME_SERVER THEN
			NonRedPointer.pbSntpServerFailuresLoc^:= TRUE;
		END_IF
	END_IF
END_IF

// Inicializa os diagnósticos locais se solicitado
IF SymbolicsNonRedundant.bEnableCleanStats_CheckSntp THEN
	NonRedPointer.pbSntpServerFailuresLoc^:= FALSE;
	NonRedPointer.pbSntpSourceFailuresLoc^:= FALSE;
	NonRedPointer.piSntpSyncFailuresLoc^:= 0;
	SymbolicsNonRedundant.bEnableCleanStats_CheckSntp:= FALSE;
END_IF

// Copia os diagnósticos locais não-redundantes para os diagnósticos persistentes redundantes
PersistentVars.bSntpServerFailures:= NonRedPointer.pbSntpServerFailuresLoc^ OR NonRedPointer.pbSntpServerFailuresRem^;
PersistentVars.bSntpSourceFailures:= NonRedPointer.pbSntpSourceFailuresLoc^ OR NonRedPointer.pbSntpSourceFailuresRem^;
IF PersistentVars.iSntpSyncFailures < ProjectConstants.iValueRedLimit THEN
	PersistentVars.iSntpSyncFailures:= NonRedPointer.piSntpSyncFailuresLoc^ + NonRedPointer.piSntpSyncFailuresRem^;
END_IF
// Registra o tempo do sistema
SysTimeGetUs(uliPouEndTime);
// Calcula duração mínima/máxima desta POU
MinMaxTimes.uliPouMinTime_CheckSntp:= MIN(MinMaxTimes.uliPouMinTime_CheckSntp, uliPouEndTime - uliPouIniTime);
MinMaxTimes.uliPouMaxTime_CheckSntp:= MAX(MinMaxTimes.uliPouMaxTime_CheckSntp, uliPouEndTime - uliPouIniTime);

END_PROGRAM

// Device/Application/UserPOUs/Non-Redundant/CheckForcing
PROGRAM CheckForcing
VAR
	bEnableCleanStatsCopy2 : BOOL;
	uliPouIniTime : ULINT;
	uliPouEndTime : ULINT;
END_VAR

// Registra o tempo do sistema
SysTimeGetUs(uliPouIniTime);

// Verifica se indicação de variável forçada está ligada
IF 	DG_NX3030.tDetailed.Application.bForcedIOs <> TRUE AND
	NonRedPointer.piForcingDiagUnsetLoc^ <= ProjectConstants.iFailCounterLimit THEN
	NonRedPointer.piForcingDiagUnsetLoc^:= NonRedPointer.piForcingDiagUnsetLoc^ + 1;
END_IF

// Verifica se variáveis que deveriam estar forçadas estão com o valor de forçamento
IF PersistentVars.bCheckForcingBoolVar <> TRUE AND
	NonRedPointer.piBoolVarNotForcedLoc^ <= ProjectConstants.iFailCounterLimit THEN
	NonRedPointer.piBoolVarNotForcedLoc^:= NonRedPointer.piBoolVarNotForcedLoc^ + 1;
END_IF
IF PersistentVars.bCheckForcingWordVar <> 12345 AND
	NonRedPointer.piWordVarNotForcedLoc^ <= ProjectConstants.iFailCounterLimit THEN
	NonRedPointer.piWordVarNotForcedLoc^:= NonRedPointer.piWordVarNotForcedLoc^ + 1;
END_IF

// Reseta o valor das variáveis que deveriam estar forçadas
PersistentVars.bCheckForcingBoolVar:= FALSE;
PersistentVars.bCheckForcingWordVar:= 0;

// Verifica solicitação de reinicialização do super teste: esta rotina deve ser
// executada depois da consistência dos forçamentos pois nos primeiros ciclos
// o diagnóstico de que existe ponto forçado ainda não está atualizado
IF SymbolicsNonRedundant.bEnableCleanStats_CheckForcing  = TRUE OR bEnableCleanStatsCopy2 = TRUE THEN
	// Reinicializa os indicadores de falha de forçamento não-redundantes
	NonRedPointer.piForcingDiagUnsetLoc^:= 0;
	NonRedPointer.piBoolVarNotForcedLoc^:= 0;
	NonRedPointer.piWordVarNotForcedLoc^:= 0;
	NonRedPointer.piForcingDiagUnsetRem^:= 0;
	NonRedPointer.piBoolVarNotForcedRem^:= 0;
	NonRedPointer.piWordVarNotForcedRem^:= 0;	
	// Garante o zeramento das variáveis de falha de forçamento por mais um ciclo,
	// visto que o diagnóstico de falha demora dois ciclos para ser atualizado
	IF SymbolicsNonRedundant.bEnableCleanStats_CheckForcing  = TRUE THEN
		bEnableCleanStatsCopy2:= TRUE;
	ELSE
		bEnableCleanStatsCopy2:= FALSE;
	END_IF
	SymbolicsNonRedundant.bEnableCleanStats_CheckForcing := FALSE;
END_IF

// Atribui as variáveis locais de falha à variáveis redundantes persistentes
	PersistentVars.bForcingDiagUnset:=	NonRedPointer.piForcingDiagUnsetLoc^ <> 0 OR
										NonRedPointer.piForcingDiagUnsetRem^ <> 0;
	PersistentVars.bBoolVarNotForced:=	NonRedPointer.piBoolVarNotForcedLoc^ <> 0 OR
										NonRedPointer.piBoolVarNotForcedRem^ <> 0;
	PersistentVars.bWordVarNotForced:=	NonRedPointer.piWordVarNotForcedLoc^ <> 0 OR
										NonRedPointer.piWordVarNotForcedRem^ <> 0;


// Registra o tempo do sistema
SysTimeGetUs(uliPouEndTime);
// Calcula duração mínima/máxima desta POU
MinMaxTimes.uliPouMinTime_CheckForcing:= MIN(MinMaxTimes.uliPouMinTime_CheckForcing, uliPouEndTime - uliPouIniTime);
MinMaxTimes.uliPouMaxTime_CheckForcing:= MAX(MinMaxTimes.uliPouMaxTime_CheckForcing, uliPouEndTime - uliPouIniTime);

END_PROGRAM

// Device/Application/UserPOUs/Non-Redundant/CheckDiagsRetain
PROGRAM CheckDiagsRetain
VAR
	bDiag_Error_NX3030 : BOOL;
	bDiag_Error_NX4010 : BOOL;
	bDiag_Error_NX5001_1 : BOOL;
	bDiag_Error_NX5001_2 : BOOL;
	bDiag_Error_NX5001_3 : BOOL;
	bDiag_Error_NX5000_1 : BOOL;
	bDiag_Error_NX5000_2 : BOOL;
	bDiag_Error_NX5000_3 : BOOL;
	bDiag_Error_MODBUS_Master_1 : BOOL;
	bDiag_Error_MODBUS_Slave_1 : BOOL;
	bDiag_Error_MODBUS_Client_2 : BOOL;
	bDiag_Error_MODBUS_Server_2 : BOOL;
	bDiag_Error_MODBUS_Client_3 : BOOL;
	bDiag_Error_MODBUS_Server_3 : BOOL;
	bDiag_Error_MODBUS_Client_4 : BOOL;
	bDiag_Error_MODBUS_Server_4 : BOOL;


	iSkipTimer : INT;
	bBoolValue : BOOL;
	dwIncrValue : DWORD;
	uliPouIniTime : ULINT;
	uliPouEndTime : ULINT;
	
	bDiag_Error_PO1000_REM05: BOOL;
	bDiag_Error_PO2020_REM05: BOOL;
	bDiag_Error_PO9100_REM05: BOOL;
	bDiag_Error_PO1212_REM10: BOOL;
	bDiag_Error_PO2132_REM10: BOOL;
	bDiag_Error_PO9100_REM10: BOOL;
	bDiag_Error_PO1000_REM04: BOOL;
	/// Depurações 1, 2 e 3
	auiDebugRedDataSync:		ARRAY[0..6] OF UINT;
	auiDebugRedForceSync:		ARRAY[0..6] OF UINT;
END_VAR

// Contadores de ciclos de diagnósticos ativos.

// Registra o tempo do sistema
SysTimeGetUs(uliPouIniTime);

// Utilizado para que alguns dos diagnósticos sejam ignorados nos primeiros ciclos como ativo 
IF DG_NX4010.tRedundancy.RedDgnLoc.sGeneral_Diag.eRedState <> REDUNDANCY_STATE.ACTIVE THEN
	// Reseta o temporizador quando não-ativo
	iSkipTimer:= iSkipTimer * 0;
ELSE
	// Mantém o temporizador inalterado quando ativo
	iSkipTimer:= iSkipTimer * 1;
END_IF

// Se já atingiu o tempo a desconsiderar os diagnósticos...
IF iSkipTimer >= ProjectConstants.iTimeToSkipAsActive THEN
	// Evita a virada do contador de ciclos
	iSkipTimer:= ProjectConstants.iTimeToSkipAsActive;
	// Irá considerar os diagnósticos em caso de falha
	bBoolValue:= TRUE;
	// Irá incrementar os diagnósticos em caso de falha
	dwIncrValue:= 1;
ELSE
	// Incrementa o temporizador como ativo
	iSkipTimer:= iSkipTimer + ProjectConstants.iMainTaskInterval;
	// Não irá considerar os diagnósticos em caso de falha
	bBoolValue:= FALSE;
	// Não irá incrementar os diagnósticos em caso de falha
	dwIncrValue:= 0;
END_IF




// NX3030
	DiagsRetain.DG_NX3030_tSummarized_bAbsentModules:= DiagsRetain.DG_NX3030_tSummarized_bAbsentModules OR DG_NX3030.tSummarized.bAbsentModules ;
	DiagsRetain.DG_NX3030_tSummarized_bAbsentRacks:= DiagsRetain.DG_NX3030_tSummarized_bAbsentRacks OR DG_NX3030.tSummarized.bAbsentRacks ;
	DiagsRetain.DG_NX3030_tSummarized_bCOM1ConfigError:= DiagsRetain.DG_NX3030_tSummarized_bCOM1ConfigError OR DG_NX3030.tSummarized.bCOM1ConfigError ;
	DiagsRetain.DG_NX3030_tSummarized_bCOM2ConfigError:= DiagsRetain.DG_NX3030_tSummarized_bCOM2ConfigError OR DG_NX3030.tSummarized.bCOM2ConfigError ;
	DiagsRetain.DG_NX3030_tSummarized_bConfigMismatch:= DiagsRetain.DG_NX3030_tSummarized_bConfigMismatch OR DG_NX3030.tSummarized.bConfigMismatch ;
	DiagsRetain.DG_NX3030_tSummarized_bDuplicatedRacks:= DiagsRetain.DG_NX3030_tSummarized_bDuplicatedRacks OR DG_NX3030.tSummarized.bDuplicatedRacks ;
	DiagsRetain.DG_NX3030_tSummarized_bDuplicatedSlots:= DiagsRetain.DG_NX3030_tSummarized_bDuplicatedSlots OR DG_NX3030.tSummarized.bDuplicatedSlots ;
	DiagsRetain.DG_NX3030_tSummarized_bHardwareFailure:= DiagsRetain.DG_NX3030_tSummarized_bHardwareFailure OR DG_NX3030.tSummarized.bHardwareFailure ;
	DiagsRetain.DG_NX3030_tSummarized_bInvalidDateTime:= DiagsRetain.DG_NX3030_tSummarized_bInvalidDateTime OR DG_NX3030.tSummarized.bInvalidDateTime ;
	DiagsRetain.DG_NX3030_tSummarized_bInvalidRacks:= DiagsRetain.DG_NX3030_tSummarized_bInvalidRacks OR DG_NX3030.tSummarized.bInvalidRacks ;
	DiagsRetain.DG_NX3030_tSummarized_bMemoryCardError:= DiagsRetain.DG_NX3030_tSummarized_bMemoryCardError OR DG_NX3030.tSummarized.bMemoryCardError ;
	DiagsRetain.DG_NX3030_tSummarized_bModuleFatalError:= DiagsRetain.DG_NX3030_tSummarized_bModuleFatalError OR DG_NX3030.tSummarized.bModuleFatalError ;
	DiagsRetain.DG_NX3030_tSummarized_bModuleParameterError:= DiagsRetain.DG_NX3030_tSummarized_bModuleParameterError OR DG_NX3030.tSummarized.bModuleParameterError ;
	DiagsRetain.DG_NX3030_tSummarized_bModulesWithDiagnostic:= DiagsRetain.DG_NX3030_tSummarized_bModulesWithDiagnostic OR (DG_NX3030.tSummarized.bModulesWithDiagnostic AND bBoolValue) ;
	DiagsRetain.DG_NX3030_tSummarized_bNET1ConfigError:= DiagsRetain.DG_NX3030_tSummarized_bNET1ConfigError OR DG_NX3030.tSummarized.bNET1ConfigError ;
	DiagsRetain.DG_NX3030_tSummarized_bNET2ConfigError:= DiagsRetain.DG_NX3030_tSummarized_bNET2ConfigError OR DG_NX3030.tSummarized.bNET2ConfigError ;
	DiagsRetain.DG_NX3030_tSummarized_bNonDeclaredModules:= DiagsRetain.DG_NX3030_tSummarized_bNonDeclaredModules OR DG_NX3030.tSummarized.bNonDeclaredModules ;
	DiagsRetain.DG_NX3030_tSummarized_bNonDeclaredRacks:= DiagsRetain.DG_NX3030_tSummarized_bNonDeclaredRacks OR DG_NX3030.tSummarized.bNonDeclaredRacks ;
	DiagsRetain.DG_NX3030_tSummarized_bOTDSwitchError:= DiagsRetain.DG_NX3030_tSummarized_bOTDSwitchError OR DG_NX3030.tSummarized.bOTDSwitchError ;
	DiagsRetain.DG_NX3030_tSummarized_bRuntimeReset:= DiagsRetain.DG_NX3030_tSummarized_bRuntimeReset OR DG_NX3030.tSummarized.bRuntimeReset ;
	DiagsRetain.DG_NX3030_tSummarized_bSoftwareException:= DiagsRetain.DG_NX3030_tSummarized_bSoftwareException OR DG_NX3030.tSummarized.bSoftwareException ;
	DiagsRetain.DG_NX3030_tSummarized_bSwappedModules:= DiagsRetain.DG_NX3030_tSummarized_bSwappedModules OR DG_NX3030.tSummarized.bSwappedModules ;
	DiagsRetain.DG_NX3030_tSummarized_bWHSBBusError:= DiagsRetain.DG_NX3030_tSummarized_bWHSBBusError OR DG_NX3030.tSummarized.bWHSBBusError ;
	DiagsRetain.DG_NX3030_tDetailed_MemoryCard_byMounted:= DiagsRetain.DG_NX3030_tDetailed_MemoryCard_byMounted OR NOT(DG_NX3030.tDetailed.MemoryCard.byMounted = MOUNTED);
	DiagsRetain.DG_NX3030_tDetailed_Ethernet_NET1_bLinkDown:= DiagsRetain.DG_NX3030_tDetailed_Ethernet_NET1_bLinkDown OR DG_NX3030.tDetailed.Ethernet.NET1.bLinkDown ;
	//DiagsRetain.DG_NX3030_tDetailed_Ethernet_NET2_bLinkDown:= DiagsRetain.DG_NX3030_tDetailed_Ethernet_NET2_bLinkDown OR DG_NX3030.tDetailed.Ethernet.NET2.bLinkDown ;
	DiagsRetain.DG_NX3030_tDetailed_Application_byCPUState	:=	DiagsRetain.DG_NX3030_tDetailed_Application_byCPUState	OR	NOT(DG_NX3030.tDetailed.Application.byCPUState = 1);
	DiagsRetain.DG_NX3030_tDetailed_ApplicationInfo_dwApplicationCRC	:=	DiagsRetain.DG_NX3030_tDetailed_ApplicationInfo_dwApplicationCRC	OR	DG_NX3030.tDetailed.ApplicationInfo.dwApplicationCRC = 0 AND FALSE;
	DiagsRetain.DG_NX3030_tDetailed_Ethernet_NET1_abyMAC_0	:=	DiagsRetain.DG_NX3030_tDetailed_Ethernet_NET1_abyMAC_0	OR	NOT(DG_NX3030.tDetailed.Ethernet.NET1.abyMAC[0] = 16#00);
	DiagsRetain.DG_NX3030_tDetailed_Ethernet_NET1_abyMAC_1	:=	DiagsRetain.DG_NX3030_tDetailed_Ethernet_NET1_abyMAC_1	OR	NOT(DG_NX3030.tDetailed.Ethernet.NET1.abyMAC[1] = 16#80);
	DiagsRetain.DG_NX3030_tDetailed_Ethernet_NET1_abyMAC_2	:=	DiagsRetain.DG_NX3030_tDetailed_Ethernet_NET1_abyMAC_2	OR	NOT(DG_NX3030.tDetailed.Ethernet.NET1.abyMAC[2] = 16#A0);
	DiagsRetain.DG_NX3030_tDetailed_Ethernet_NET1_abyMAC_3	:=	DiagsRetain.DG_NX3030_tDetailed_Ethernet_NET1_abyMAC_3	OR	NOT(DG_NX3030.tDetailed.Ethernet.NET1.abyMAC[3] = 16#05);
	DiagsRetain.DG_NX3030_tDetailed_Ethernet_NET1_abyMAC_4	:=	DiagsRetain.DG_NX3030_tDetailed_Ethernet_NET1_abyMAC_4	OR	NOT(DG_NX3030.tDetailed.Ethernet.NET1.abyMAC[4] = 16#F1);
	DiagsRetain.DG_NX3030_tDetailed_Ethernet_NET1_abyMAC_5	:=	DiagsRetain.DG_NX3030_tDetailed_Ethernet_NET1_abyMAC_5	OR	NOT(DG_NX3030.tDetailed.Ethernet.NET1.abyMAC[5] = 16#84 OR DG_NX3030.tDetailed.Ethernet.NET1.abyMAC[5] = 16#98);
	DiagsRetain.DG_NX3030_tDetailed_Ethernet_NET2_abyMAC_0	:=	DiagsRetain.DG_NX3030_tDetailed_Ethernet_NET2_abyMAC_0	OR	NOT(DG_NX3030.tDetailed.Ethernet.NET2.abyMAC[0] = 16#00);
	DiagsRetain.DG_NX3030_tDetailed_Ethernet_NET2_abyMAC_1	:=	DiagsRetain.DG_NX3030_tDetailed_Ethernet_NET2_abyMAC_1	OR	NOT(DG_NX3030.tDetailed.Ethernet.NET2.abyMAC[1] = 16#80);
	DiagsRetain.DG_NX3030_tDetailed_Ethernet_NET2_abyMAC_2	:=	DiagsRetain.DG_NX3030_tDetailed_Ethernet_NET2_abyMAC_2	OR	NOT(DG_NX3030.tDetailed.Ethernet.NET2.abyMAC[2] = 16#A0);
	DiagsRetain.DG_NX3030_tDetailed_Ethernet_NET2_abyMAC_3	:=	DiagsRetain.DG_NX3030_tDetailed_Ethernet_NET2_abyMAC_3	OR	NOT(DG_NX3030.tDetailed.Ethernet.NET2.abyMAC[3] = 16#05);
	DiagsRetain.DG_NX3030_tDetailed_Ethernet_NET2_abyMAC_4	:=	DiagsRetain.DG_NX3030_tDetailed_Ethernet_NET2_abyMAC_4	OR	NOT(DG_NX3030.tDetailed.Ethernet.NET2.abyMAC[4] = 16#F1);
	DiagsRetain.DG_NX3030_tDetailed_Ethernet_NET2_abyMAC_5	:=	DiagsRetain.DG_NX3030_tDetailed_Ethernet_NET2_abyMAC_5	OR	NOT(DG_NX3030.tDetailed.Ethernet.NET2.abyMAC[5] = 16#85 OR DG_NX3030.tDetailed.Ethernet.NET2.abyMAC[5] = 16#99);
	DiagsRetain.DG_NX3030_tDetailed_Ethernet_NETx_abyIP_0	:=	DiagsRetain.DG_NX3030_tDetailed_Ethernet_NETx_abyIP_0	OR	NOT(DG_NX3030.tDetailed.Ethernet.NET1.abyIP[0] = 192 OR DG_NX3030.tDetailed.Ethernet.NET2.abyIP[0] = 192);
	DiagsRetain.DG_NX3030_tDetailed_Ethernet_NETx_abyIP_1	:=	DiagsRetain.DG_NX3030_tDetailed_Ethernet_NETx_abyIP_1	OR	NOT(DG_NX3030.tDetailed.Ethernet.NET1.abyIP[1] = 168 OR DG_NX3030.tDetailed.Ethernet.NET2.abyIP[1] = 168);
	DiagsRetain.DG_NX3030_tDetailed_Ethernet_NETx_abyIP_2	:=	DiagsRetain.DG_NX3030_tDetailed_Ethernet_NETx_abyIP_2	OR	NOT(DG_NX3030.tDetailed.Ethernet.NET1.abyIP[2] = 23 OR DG_NX3030.tDetailed.Ethernet.NET2.abyIP[2] = 23);
	DiagsRetain.DG_NX3030_tDetailed_Ethernet_NETx_abyIP_3	:=	DiagsRetain.DG_NX3030_tDetailed_Ethernet_NETx_abyIP_3	OR	NOT(DG_NX3030.tDetailed.Ethernet.NET1.abyIP[3] = 1 OR DG_NX3030.tDetailed.Ethernet.NET2.abyIP[3] = 1 OR DG_NX3030.tDetailed.Ethernet.NET1.abyIP[3] = 2 OR DG_NX3030.tDetailed.Ethernet.NET2.abyIP[3] = 2);
	DiagsRetain.DG_NX3030_tDetailed_Ethernet_NETx_abyMask_0	:=	DiagsRetain.DG_NX3030_tDetailed_Ethernet_NETx_abyMask_0	OR	NOT(DG_NX3030.tDetailed.Ethernet.NET1.abyMASK[0] = 255 OR DG_NX3030.tDetailed.Ethernet.NET2.abyMASK[0] = 255);
	DiagsRetain.DG_NX3030_tDetailed_Ethernet_NETx_abyMask_1	:=	DiagsRetain.DG_NX3030_tDetailed_Ethernet_NETx_abyMask_1	OR	NOT(DG_NX3030.tDetailed.Ethernet.NET1.abyMASK[1] = 255 OR DG_NX3030.tDetailed.Ethernet.NET2.abyMASK[1] = 255);
	DiagsRetain.DG_NX3030_tDetailed_Ethernet_NETx_abyMask_2	:=	DiagsRetain.DG_NX3030_tDetailed_Ethernet_NETx_abyMask_2	OR	NOT(DG_NX3030.tDetailed.Ethernet.NET1.abyMASK[2] = 248 OR DG_NX3030.tDetailed.Ethernet.NET2.abyMASK[2] = 248);
	DiagsRetain.DG_NX3030_tDetailed_Ethernet_NETx_abyMask_3	:=	DiagsRetain.DG_NX3030_tDetailed_Ethernet_NETx_abyMask_3	OR	NOT(DG_NX3030.tDetailed.Ethernet.NET1.abyMASK[3] = 0 OR DG_NX3030.tDetailed.Ethernet.NET2.abyMASK[3] = 0);
	DiagsRetain.DG_NX3030_tDetailed_Ethernet_NETx_abyGateway_0	:=	DiagsRetain.DG_NX3030_tDetailed_Ethernet_NETx_abyGateway_0	OR	NOT(DG_NX3030.tDetailed.Ethernet.NET1.abyGateWAY[0] = 192 OR DG_NX3030.tDetailed.Ethernet.NET2.abyGateWAY[0] = 192);
	DiagsRetain.DG_NX3030_tDetailed_Ethernet_NETx_abyGateway_1	:=	DiagsRetain.DG_NX3030_tDetailed_Ethernet_NETx_abyGateway_1	OR	NOT(DG_NX3030.tDetailed.Ethernet.NET1.abyGateWAY[1] = 168 OR DG_NX3030.tDetailed.Ethernet.NET2.abyGateWAY[1] = 168);
	DiagsRetain.DG_NX3030_tDetailed_Ethernet_NETx_abyGateway_2	:=	DiagsRetain.DG_NX3030_tDetailed_Ethernet_NETx_abyGateway_2	OR	NOT(DG_NX3030.tDetailed.Ethernet.NET1.abyGateWAY[2] = 16 OR DG_NX3030.tDetailed.Ethernet.NET2.abyGateWAY[2] = 16);
	DiagsRetain.DG_NX3030_tDetailed_Ethernet_NETx_abyGateway_3	:=	DiagsRetain.DG_NX3030_tDetailed_Ethernet_NETx_abyGateway_3	OR	NOT(DG_NX3030.tDetailed.Ethernet.NET1.abyGateWAY[3] = 253 OR DG_NX3030.tDetailed.Ethernet.NET2.abyGateWAY[3] = 253);
	DiagsRetain.DG_NX3030_tDetailed_SNTP_bServiceEnabled	:=	DiagsRetain.DG_NX3030_tDetailed_SNTP_bServiceEnabled	OR	NOT(DG_NX3030.tDetailed.SNTP.bServiceEnabled =  TRUE);
	DiagsRetain.DG_NX3030_tDetailed_Target_abyAuxprocVersion	:=	DiagsRetain.DG_NX3030_tDetailed_Target_abyAuxprocVersion	OR	(DG_NX3030.tDetailed.Target.abyAuxprocVersion[0] = 0 AND 
																											 DG_NX3030.tDetailed.Target.abyAuxprocVersion[1] = 0 AND 
																											 DG_NX3030.tDetailed.Target.abyAuxprocVersion[2] = 0 AND	
																											 DG_NX3030.tDetailed.Target.abyAuxprocVersion[3] = 0);	
	DiagsRetain.DG_NX3030_tDetailed_Target_abyBootloaderVersion	:=	DiagsRetain.DG_NX3030_tDetailed_Target_abyBootloaderVersion	OR	(DG_NX3030.tDetailed.Target.abyBootloaderVersion[0] = 0 AND	
																											 DG_NX3030.tDetailed.Target.abyBootloaderVersion[1] = 0 AND	
																											 DG_NX3030.tDetailed.Target.abyBootloaderVersion[2] = 0 AND	
																											 DG_NX3030.tDetailed.Target.abyBootloaderVersion[3] = 0);	
	DiagsRetain.DG_NX3030_tDetailed_Target_abyCPUVersion	:=	DiagsRetain.DG_NX3030_tDetailed_Target_abyCPUVersion	OR	(DG_NX3030.tDetailed.Target.abyCPUVersion[0] = 0 AND		
																									 DG_NX3030.tDetailed.Target.abyCPUVersion[1] = 0 AND	
																									 DG_NX3030.tDetailed.Target.abyCPUVersion[2] = 0 AND	
																									 DG_NX3030.tDetailed.Target.abyCPUVersion[3] = 0);	
	DiagsRetain.DG_NX3030_tDetailed_Target_dwCPUModel	:=	DiagsRetain.DG_NX3030_tDetailed_Target_dwCPUModel	OR	NOT(DG_NX3030.tDetailed.Target.dwCPUModel = 16#3030);
	DiagsRetain.DG_NX3030_tDetailed_Thermometer_diTemperature	:=	DiagsRetain.DG_NX3030_tDetailed_Thermometer_diTemperature	OR	DG_NX3030.tDetailed.Thermometer.diTemperature = 0;

	
// NX4010
	DiagsRetain.DG_NX4010_tGeneral_bActiveDiagnostics:= DiagsRetain.DG_NX4010_tGeneral_bActiveDiagnostics OR DG_NX4010.tGeneral.bActiveDiagnostics ;
	DiagsRetain.DG_NX4010_tGeneral_bBusCommunicationError:= DiagsRetain.DG_NX4010_tGeneral_bBusCommunicationError OR DG_NX4010.tGeneral.bBusCommunicationError ;
	DiagsRetain.DG_NX4010_tGeneral_bConfigMismatch:= DiagsRetain.DG_NX4010_tGeneral_bConfigMismatch OR DG_NX4010.tGeneral.bConfigMismatch ;
	DiagsRetain.DG_NX4010_tGeneral_bFatalError:= DiagsRetain.DG_NX4010_tGeneral_bFatalError OR DG_NX4010.tGeneral.bFatalError ;
	DiagsRetain.DG_NX4010_tGeneral_bNET1LinkDown:= DiagsRetain.DG_NX4010_tGeneral_bNET1LinkDown OR DG_NX4010.tGeneral.bNET1LinkDown ;
	DiagsRetain.DG_NX4010_tGeneral_bNET2LinkDown:= DiagsRetain.DG_NX4010_tGeneral_bNET2LinkDown OR DG_NX4010.tGeneral.bNET2LinkDown ;
	DiagsRetain.DG_NX4010_tGeneral_bOTDSwitchError:= DiagsRetain.DG_NX4010_tGeneral_bOTDSwitchError OR DG_NX4010.tGeneral.bOTDSwitchError ;
	DiagsRetain.DG_NX4010_tGeneral_bWatchdogError:= DiagsRetain.DG_NX4010_tGeneral_bWatchdogError OR DG_NX4010.tGeneral.bWatchdogError ;
	DiagsRetain.DG_NX4010_tRedundancy_RedDgnLoc_sGeneral_Diag_bApplicationIncompatible:= DiagsRetain.DG_NX4010_tRedundancy_RedDgnLoc_sGeneral_Diag_bApplicationIncompatible OR DG_NX4010.tRedundancy.RedDgnLoc.sGeneral_Diag.bApplicationIncompatible ;
	DiagsRetain.DG_NX4010_tRedundancy_RedDgnLoc_sGeneral_Diag_bApplicationProjectDiff:= DiagsRetain.DG_NX4010_tRedundancy_RedDgnLoc_sGeneral_Diag_bApplicationProjectDiff OR DG_NX4010.tRedundancy.RedDgnLoc.sGeneral_Diag.bApplicationProjectDiff ;
	DiagsRetain.DG_NX4010_tRedundancy_RedDgnLoc_sGeneral_Diag_bConfigError:= DiagsRetain.DG_NX4010_tRedundancy_RedDgnLoc_sGeneral_Diag_bConfigError OR DG_NX4010.tRedundancy.RedDgnLoc.sGeneral_Diag.bConfigError ;
	DiagsRetain.DG_NX4010_tRedundancy_RedDgnLoc_sGeneral_Diag_bExchangeSync:= DiagsRetain.DG_NX4010_tRedundancy_RedDgnLoc_sGeneral_Diag_bExchangeSync OR NOT DG_NX4010.tRedundancy.RedDgnLoc.sGeneral_Diag.bExchangeSync ;
	DiagsRetain.DG_NX4010_tRedundancy_RedDgnLoc_sGeneral_Diag_bFailedPBUS1A:= DiagsRetain.DG_NX4010_tRedundancy_RedDgnLoc_sGeneral_Diag_bFailedPBUS1A OR DG_NX4010.tRedundancy.RedDgnLoc.sGeneral_Diag.bFailedPBUS1A ;
	DiagsRetain.DG_NX4010_tRedundancy_RedDgnLoc_sGeneral_Diag_bFailedPBUS1B:= DiagsRetain.DG_NX4010_tRedundancy_RedDgnLoc_sGeneral_Diag_bFailedPBUS1B OR DG_NX4010.tRedundancy.RedDgnLoc.sGeneral_Diag.bFailedPBUS1B ;
	DiagsRetain.DG_NX4010_tRedundancy_RedDgnLoc_sGeneral_Diag_bFailedPBUS2A:= DiagsRetain.DG_NX4010_tRedundancy_RedDgnLoc_sGeneral_Diag_bFailedPBUS2A OR DG_NX4010.tRedundancy.RedDgnLoc.sGeneral_Diag.bFailedPBUS2A ;
	DiagsRetain.DG_NX4010_tRedundancy_RedDgnLoc_sGeneral_Diag_bFailedPBUS2B:= DiagsRetain.DG_NX4010_tRedundancy_RedDgnLoc_sGeneral_Diag_bFailedPBUS2B OR DG_NX4010.tRedundancy.RedDgnLoc.sGeneral_Diag.bFailedPBUS2B ;
	DiagsRetain.DG_NX4010_tRedundancy_RedDgnLoc_sGeneral_Diag_bFailedRED:= DiagsRetain.DG_NX4010_tRedundancy_RedDgnLoc_sGeneral_Diag_bFailedRED OR DG_NX4010.tRedundancy.RedDgnLoc.sGeneral_Diag.bFailedRED ;
	DiagsRetain.DG_NX4010_tRedundancy_RedDgnLoc_sGeneral_Diag_bFailureProfibus_1:= DiagsRetain.DG_NX4010_tRedundancy_RedDgnLoc_sGeneral_Diag_bFailureProfibus_1 OR DG_NX4010.tRedundancy.RedDgnLoc.sGeneral_Diag.bFailureProfibus_1 ;
	DiagsRetain.DG_NX4010_tRedundancy_RedDgnLoc_sGeneral_Diag_bFailureProfibus_2:= DiagsRetain.DG_NX4010_tRedundancy_RedDgnLoc_sGeneral_Diag_bFailureProfibus_2 OR DG_NX4010.tRedundancy.RedDgnLoc.sGeneral_Diag.bFailureProfibus_2 ;
	DiagsRetain.DG_NX4010_tRedundancy_RedDgnLoc_sGeneral_Diag_bIncompatibleFirmware:= DiagsRetain.DG_NX4010_tRedundancy_RedDgnLoc_sGeneral_Diag_bIncompatibleFirmware OR DG_NX4010.tRedundancy.RedDgnLoc.sGeneral_Diag.bIncompatibleFirmware ;
	DiagsRetain.DG_NX4010_tRedundancy_RedDgnLoc_sGeneral_Diag_bProfibusVitalFailureAll:= DiagsRetain.DG_NX4010_tRedundancy_RedDgnLoc_sGeneral_Diag_bProfibusVitalFailureAll OR DG_NX4010.tRedundancy.RedDgnLoc.sGeneral_Diag.bProfibusVitalFailureAll ;
	DiagsRetain.DG_NX4010_tRedundancy_RedDgnLoc_sGeneral_Diag_bProfibusVitalFailureAny:= DiagsRetain.DG_NX4010_tRedundancy_RedDgnLoc_sGeneral_Diag_bProfibusVitalFailureAny OR DG_NX4010.tRedundancy.RedDgnLoc.sGeneral_Diag.bProfibusVitalFailureAny ;
	DiagsRetain.DG_NX4010_tRedundancy_RedDgnLoc_sGeneral_Diag_bProjectArchiveDiff:= DiagsRetain.DG_NX4010_tRedundancy_RedDgnLoc_sGeneral_Diag_bProjectArchiveDiff OR DG_NX4010.tRedundancy.RedDgnLoc.sGeneral_Diag.bProjectArchiveDiff ;
	DiagsRetain.DG_NX4010_tRedundancy_RedDgnLoc_sGeneral_Diag_bProjectSyncDisable:= DiagsRetain.DG_NX4010_tRedundancy_RedDgnLoc_sGeneral_Diag_bProjectSyncDisable OR DG_NX4010.tRedundancy.RedDgnLoc.sGeneral_Diag.bProjectSyncDisable ;
	DiagsRetain.DG_NX4010_tRedundancy_RedDgnLoc_sGeneral_Diag_bRedDataSync:= DiagsRetain.DG_NX4010_tRedundancy_RedDgnLoc_sGeneral_Diag_bRedDataSync OR NOT DG_NX4010.tRedundancy.RedDgnLoc.sGeneral_Diag.bRedDataSync ;
	DiagsRetain.DG_NX4010_tRedundancy_RedDgnLoc_sGeneral_Diag_bRedForceSync:= DiagsRetain.DG_NX4010_tRedundancy_RedDgnLoc_sGeneral_Diag_bRedForceSync OR NOT DG_NX4010.tRedundancy.RedDgnLoc.sGeneral_Diag.bRedForceSync ;
	DiagsRetain.DG_NX4010_tRedundancy_RedDgnLoc_sGeneral_Diag_bRedPanelTestMode:= DiagsRetain.DG_NX4010_tRedundancy_RedDgnLoc_sGeneral_Diag_bRedPanelTestMode OR DG_NX4010.tRedundancy.RedDgnLoc.sGeneral_Diag.bRedPanelTestMode ;
	DiagsRetain.DG_NX4010_tRedundancy_RedDgnLoc_sGeneral_Diag_bTemporaryBufferTooSmall:= DiagsRetain.DG_NX4010_tRedundancy_RedDgnLoc_sGeneral_Diag_bTemporaryBufferTooSmall OR DG_NX4010.tRedundancy.RedDgnLoc.sGeneral_Diag.bTemporaryBufferTooSmall ;
	DiagsRetain.DG_NX4010_tRedundancy_RedDgnLoc_sGeneral_Diag_bTooManyRedAreas:= DiagsRetain.DG_NX4010_tRedundancy_RedDgnLoc_sGeneral_Diag_bTooManyRedAreas OR DG_NX4010.tRedundancy.RedDgnLoc.sGeneral_Diag.bTooManyRedAreas ;
	DiagsRetain.DG_NX4010_tRedundancy_RedDgnLoc_sGeneral_Diag_dwApplicationCRC:= DiagsRetain.DG_NX4010_tRedundancy_RedDgnLoc_sGeneral_Diag_dwApplicationCRC OR DG_NX4010.tRedundancy.RedDgnLoc.sGeneral_Diag.dwApplicationCRC = 16#FFFFFFFF;
	DiagsRetain.DG_NX4010_tRedundancy_RedDgnLoc_sGeneral_Diag_dwArchiveCRC:= DiagsRetain.DG_NX4010_tRedundancy_RedDgnLoc_sGeneral_Diag_dwArchiveCRC OR DG_NX4010.tRedundancy.RedDgnLoc.sGeneral_Diag.dwArchiveCRC = 16#FFFFFFFF;
	
// NX5001_1
	DiagsRetain.DG_NX5001_1_tGeneral_bActiveDiagnostics:= DiagsRetain.DG_NX5001_1_tGeneral_bActiveDiagnostics OR (DG_NX5001_1.tGeneral.bActiveDiagnostics AND bBoolValue) ;
	DiagsRetain.DG_NX5001_1_tGeneral_bBusCommunicationError:= DiagsRetain.DG_NX5001_1_tGeneral_bBusCommunicationError OR DG_NX5001_1.tGeneral.bBusCommunicationError ;
	DiagsRetain.DG_NX5001_1_tGeneral_bConfigMismatch:= DiagsRetain.DG_NX5001_1_tGeneral_bConfigMismatch OR DG_NX5001_1.tGeneral.bConfigMismatch ;
	DiagsRetain.DG_NX5001_1_tGeneral_bFatalError:= DiagsRetain.DG_NX5001_1_tGeneral_bFatalError OR DG_NX5001_1.tGeneral.bFatalError ;
	DiagsRetain.DG_NX5001_1_tGeneral_bNX5001NoCfg:= DiagsRetain.DG_NX5001_1_tGeneral_bNX5001NoCfg OR DG_NX5001_1.tGeneral.bNX5001NoCfg ;
	DiagsRetain.DG_NX5001_1_tGeneral_bOTDSwitchError:= DiagsRetain.DG_NX5001_1_tGeneral_bOTDSwitchError OR DG_NX5001_1.tGeneral.bOTDSwitchError ;
	DiagsRetain.DG_NX5001_1_tGeneral_bPbusCommFail:= DiagsRetain.DG_NX5001_1_tGeneral_bPbusCommFail OR (DG_NX5001_1.tGeneral.bPbusCommFail AND bBoolValue) ;
	DiagsRetain.DG_NX5001_1_tGeneral_bSlaveNotConfigured:= DiagsRetain.DG_NX5001_1_tGeneral_bSlaveNotConfigured OR (DG_NX5001_1.tGeneral.bSlaveNotConfigured AND bBoolValue) ;
	DiagsRetain.DG_NX5001_1_tGeneral_bSlaveNotPresent:= DiagsRetain.DG_NX5001_1_tGeneral_bSlaveNotPresent OR DG_NX5001_1.tGeneral.bSlaveNotPresent ;
	DiagsRetain.DG_NX5001_1_tGeneral_bSlaveWithDiagnostic:= DiagsRetain.DG_NX5001_1_tGeneral_bSlaveWithDiagnostic OR DG_NX5001_1.tGeneral.bSlaveWithDiagnostic ;
	DiagsRetain.DG_NX5001_1_tGeneral_bStsEnableInterface:= DiagsRetain.DG_NX5001_1_tGeneral_bStsEnableInterface OR (NOT DG_NX5001_1.tGeneral.bStsEnableInterface AND bBoolValue) ;
	DiagsRetain.DG_NX5001_1_tGeneral_bStsMstRedundEnable:= DiagsRetain.DG_NX5001_1_tGeneral_bStsMstRedundEnable OR NOT DG_NX5001_1.tGeneral.bStsMstRedundEnable ;
	DiagsRetain.DG_NX5001_1_tGeneral_bWatchdogError:= DiagsRetain.DG_NX5001_1_tGeneral_bWatchdogError OR DG_NX5001_1.tGeneral.bWatchdogError ;
	DiagsRetain.DG_NX5001_1_tMstStatus_abySlv_Diag_bSlave_5:= DiagsRetain.DG_NX5001_1_tMstStatus_abySlv_Diag_bSlave_5 OR DG_NX5001_1.tMstStatus.abySlv_Diag.bSlave_5;
	DiagsRetain.DG_NX5001_1_tMstStatus_abySlv_Diag_bSlave_10:= DiagsRetain.DG_NX5001_1_tMstStatus_abySlv_Diag_bSlave_10 OR DG_NX5001_1.tMstStatus.abySlv_Diag.bSlave_10;
	
// NX5001_2
	DiagsRetain.DG_NX5001_2_tGeneral_bActiveDiagnostics:= DiagsRetain.DG_NX5001_2_tGeneral_bActiveDiagnostics OR (DG_NX5001_2.tGeneral.bActiveDiagnostics AND bBoolValue);
	DiagsRetain.DG_NX5001_2_tGeneral_bBusCommunicationError:= DiagsRetain.DG_NX5001_2_tGeneral_bBusCommunicationError OR DG_NX5001_2.tGeneral.bBusCommunicationError ;
	DiagsRetain.DG_NX5001_2_tGeneral_bConfigMismatch:= DiagsRetain.DG_NX5001_2_tGeneral_bConfigMismatch OR DG_NX5001_2.tGeneral.bConfigMismatch ;
	DiagsRetain.DG_NX5001_2_tGeneral_bFatalError:= DiagsRetain.DG_NX5001_2_tGeneral_bFatalError OR DG_NX5001_2.tGeneral.bFatalError ;
	DiagsRetain.DG_NX5001_2_tGeneral_bNX5001NoCfg:= DiagsRetain.DG_NX5001_2_tGeneral_bNX5001NoCfg OR DG_NX5001_2.tGeneral.bNX5001NoCfg ;
	DiagsRetain.DG_NX5001_2_tGeneral_bOTDSwitchError:= DiagsRetain.DG_NX5001_2_tGeneral_bOTDSwitchError OR DG_NX5001_2.tGeneral.bOTDSwitchError ;
	DiagsRetain.DG_NX5001_2_tGeneral_bPbusCommFail:= DiagsRetain.DG_NX5001_2_tGeneral_bPbusCommFail OR (DG_NX5001_2.tGeneral.bPbusCommFail AND bBoolValue) ;
	DiagsRetain.DG_NX5001_2_tGeneral_bSlaveNotConfigured:= DiagsRetain.DG_NX5001_2_tGeneral_bSlaveNotConfigured OR (DG_NX5001_2.tGeneral.bSlaveNotConfigured AND bBoolValue) ;
	DiagsRetain.DG_NX5001_2_tGeneral_bSlaveNotPresent:= DiagsRetain.DG_NX5001_2_tGeneral_bSlaveNotPresent OR DG_NX5001_2.tGeneral.bSlaveNotPresent ;
	DiagsRetain.DG_NX5001_2_tGeneral_bSlaveWithDiagnostic:= DiagsRetain.DG_NX5001_2_tGeneral_bSlaveWithDiagnostic OR DG_NX5001_2.tGeneral.bSlaveWithDiagnostic ;
	DiagsRetain.DG_NX5001_2_tGeneral_bStsEnableInterface:= DiagsRetain.DG_NX5001_2_tGeneral_bStsEnableInterface OR (NOT DG_NX5001_2.tGeneral.bStsEnableInterface AND bBoolValue) ;
	DiagsRetain.DG_NX5001_2_tGeneral_bStsMstRedundEnable:= DiagsRetain.DG_NX5001_2_tGeneral_bStsMstRedundEnable OR  NOT DG_NX5001_2.tGeneral.bStsMstRedundEnable ;
	DiagsRetain.DG_NX5001_2_tGeneral_bWatchdogError:= DiagsRetain.DG_NX5001_2_tGeneral_bWatchdogError OR DG_NX5001_2.tGeneral.bWatchdogError ;
	DiagsRetain.DG_NX5001_2_tMstStatus_abySlv_Diag_bSlave_5:= DiagsRetain.DG_NX5001_2_tMstStatus_abySlv_Diag_bSlave_5 OR DG_NX5001_2.tMstStatus.abySlv_Diag.bSlave_5;
	DiagsRetain.DG_NX5001_2_tMstStatus_abySlv_Diag_bSlave_10:= DiagsRetain.DG_NX5001_2_tMstStatus_abySlv_Diag_bSlave_10 OR DG_NX5001_2.tMstStatus.abySlv_Diag.bSlave_10;

// NX5001_3
	DiagsRetain.DG_NX5001_3_tGeneral_bActiveDiagnostics:= DiagsRetain.DG_NX5001_3_tGeneral_bActiveDiagnostics OR (DG_NX5001_3.tGeneral.bActiveDiagnostics AND bBoolValue) ;
	DiagsRetain.DG_NX5001_3_tGeneral_bBusCommunicationError:= DiagsRetain.DG_NX5001_3_tGeneral_bBusCommunicationError OR DG_NX5001_3.tGeneral.bBusCommunicationError ;
	DiagsRetain.DG_NX5001_3_tGeneral_bConfigMismatch:= DiagsRetain.DG_NX5001_3_tGeneral_bConfigMismatch OR DG_NX5001_3.tGeneral.bConfigMismatch ;
	DiagsRetain.DG_NX5001_3_tGeneral_bFatalError:= DiagsRetain.DG_NX5001_3_tGeneral_bFatalError OR DG_NX5001_3.tGeneral.bFatalError ;
	DiagsRetain.DG_NX5001_3_tGeneral_bNX5001NoCfg:= DiagsRetain.DG_NX5001_3_tGeneral_bNX5001NoCfg OR DG_NX5001_3.tGeneral.bNX5001NoCfg ;
	DiagsRetain.DG_NX5001_3_tGeneral_bOTDSwitchError:= DiagsRetain.DG_NX5001_3_tGeneral_bOTDSwitchError OR DG_NX5001_3.tGeneral.bOTDSwitchError ;
	DiagsRetain.DG_NX5001_3_tGeneral_bPbusCommFail:= DiagsRetain.DG_NX5001_3_tGeneral_bPbusCommFail OR (DG_NX5001_3.tGeneral.bPbusCommFail AND bBoolValue) ;
	DiagsRetain.DG_NX5001_3_tGeneral_bSlaveNotConfigured:= DiagsRetain.DG_NX5001_3_tGeneral_bSlaveNotConfigured OR (DG_NX5001_3.tGeneral.bSlaveNotConfigured AND bBoolValue) ;
	DiagsRetain.DG_NX5001_3_tGeneral_bSlaveNotPresent:= DiagsRetain.DG_NX5001_3_tGeneral_bSlaveNotPresent OR DG_NX5001_3.tGeneral.bSlaveNotPresent ;
	DiagsRetain.DG_NX5001_3_tGeneral_bSlaveWithDiagnostic:= DiagsRetain.DG_NX5001_3_tGeneral_bSlaveWithDiagnostic OR DG_NX5001_3.tGeneral.bSlaveWithDiagnostic ;
	DiagsRetain.DG_NX5001_3_tGeneral_bStsEnableInterface:= DiagsRetain.DG_NX5001_3_tGeneral_bStsEnableInterface OR (NOT DG_NX5001_3.tGeneral.bStsEnableInterface AND bBoolValue) ;
	DiagsRetain.DG_NX5001_3_tGeneral_bStsMstRedundEnable:= DiagsRetain.DG_NX5001_3_tGeneral_bStsMstRedundEnable OR NOT DG_NX5001_3.tGeneral.bStsMstRedundEnable ;
	DiagsRetain.DG_NX5001_3_tGeneral_bWatchdogError:= DiagsRetain.DG_NX5001_3_tGeneral_bWatchdogError OR DG_NX5001_3.tGeneral.bWatchdogError ;
	DiagsRetain.DG_NX5001_3_tMstStatus_abySlv_Diag_bSlave_4:= DiagsRetain.DG_NX5001_3_tMstStatus_abySlv_Diag_bSlave_4 OR DG_NX5001_3.tMstStatus.abySlv_Diag.bSlave_4;
	DiagsRetain.DG_NX5001_3_tMstStatus_abySlv_Diag_bSlave_99:= DiagsRetain.DG_NX5001_3_tMstStatus_abySlv_Diag_bSlave_99 OR DG_NX5001_3.tMstStatus.abySlv_Diag.bSlave_99;
	
// NX5000_1	
 	DiagsRetain.DG_NX5000_1_tGeneral_bActiveDiagnostics:= DiagsRetain.DG_NX5000_1_tGeneral_bActiveDiagnostics OR DG_NX5000_1.tGeneral.bActiveDiagnostics ;
	DiagsRetain.DG_NX5000_1_tGeneral_bBusCommunicationError:= DiagsRetain.DG_NX5000_1_tGeneral_bBusCommunicationError OR DG_NX5000_1.tGeneral.bBusCommunicationError ;
	DiagsRetain.DG_NX5000_1_tGeneral_bConfigMismatch:= DiagsRetain.DG_NX5000_1_tGeneral_bConfigMismatch OR DG_NX5000_1.tGeneral.bConfigMismatch ;
	DiagsRetain.DG_NX5000_1_tGeneral_bFatalError:= DiagsRetain.DG_NX5000_1_tGeneral_bFatalError OR DG_NX5000_1.tGeneral.bFatalError ;
	DiagsRetain.DG_NX5000_1_tGeneral_bOTDSwitchError:= DiagsRetain.DG_NX5000_1_tGeneral_bOTDSwitchError OR DG_NX5000_1.tGeneral.bOTDSwitchError ;
	DiagsRetain.DG_NX5000_1_tGeneral_bWatchdogError:= DiagsRetain.DG_NX5000_1_tGeneral_bWatchdogError OR DG_NX5000_1.tGeneral.bWatchdogError ;
	DiagsRetain.DG_NX5000_1_tNX5000_bNX5000NoCfg:= DiagsRetain.DG_NX5000_1_tNX5000_bNX5000NoCfg OR DG_NX5000_1.tNX5000.bNX5000NoCfg ;
	DiagsRetain.DG_NX5000_1_tNX5000_bStsEthLink:= DiagsRetain.DG_NX5000_1_tNX5000_bStsEthLink OR DG_NX5000_1.tNX5000.bStsEthLink ;	

// NX5000_2	
 	DiagsRetain.DG_NX5000_2_tGeneral_bActiveDiagnostics:= DiagsRetain.DG_NX5000_2_tGeneral_bActiveDiagnostics OR DG_NX5000_2.tGeneral.bActiveDiagnostics ;
	DiagsRetain.DG_NX5000_2_tGeneral_bBusCommunicationError:= DiagsRetain.DG_NX5000_2_tGeneral_bBusCommunicationError OR DG_NX5000_2.tGeneral.bBusCommunicationError ;
	DiagsRetain.DG_NX5000_2_tGeneral_bConfigMismatch:= DiagsRetain.DG_NX5000_2_tGeneral_bConfigMismatch OR DG_NX5000_2.tGeneral.bConfigMismatch ;
	DiagsRetain.DG_NX5000_2_tGeneral_bFatalError:= DiagsRetain.DG_NX5000_2_tGeneral_bFatalError OR DG_NX5000_2.tGeneral.bFatalError ;
	DiagsRetain.DG_NX5000_2_tGeneral_bOTDSwitchError:= DiagsRetain.DG_NX5000_2_tGeneral_bOTDSwitchError OR DG_NX5000_2.tGeneral.bOTDSwitchError ;
	DiagsRetain.DG_NX5000_2_tGeneral_bWatchdogError:= DiagsRetain.DG_NX5000_2_tGeneral_bWatchdogError OR DG_NX5000_2.tGeneral.bWatchdogError ;
	DiagsRetain.DG_NX5000_2_tNX5000_bNX5000NoCfg:= DiagsRetain.DG_NX5000_2_tNX5000_bNX5000NoCfg OR DG_NX5000_2.tNX5000.bNX5000NoCfg ;
	DiagsRetain.DG_NX5000_2_tNX5000_bStsEthLink:= DiagsRetain.DG_NX5000_2_tNX5000_bStsEthLink OR DG_NX5000_2.tNX5000.bStsEthLink ;		
	
// NX5000_3	
 	DiagsRetain.DG_NX5000_3_tGeneral_bActiveDiagnostics:= DiagsRetain.DG_NX5000_3_tGeneral_bActiveDiagnostics OR DG_NX5000_3.tGeneral.bActiveDiagnostics ;
	DiagsRetain.DG_NX5000_3_tGeneral_bBusCommunicationError:= DiagsRetain.DG_NX5000_3_tGeneral_bBusCommunicationError OR DG_NX5000_3.tGeneral.bBusCommunicationError ;
	DiagsRetain.DG_NX5000_3_tGeneral_bConfigMismatch:= DiagsRetain.DG_NX5000_3_tGeneral_bConfigMismatch OR DG_NX5000_3.tGeneral.bConfigMismatch ;
	DiagsRetain.DG_NX5000_3_tGeneral_bFatalError:= DiagsRetain.DG_NX5000_3_tGeneral_bFatalError OR DG_NX5000_3.tGeneral.bFatalError ;
	DiagsRetain.DG_NX5000_3_tGeneral_bOTDSwitchError:= DiagsRetain.DG_NX5000_3_tGeneral_bOTDSwitchError OR DG_NX5000_3.tGeneral.bOTDSwitchError ;
	DiagsRetain.DG_NX5000_3_tGeneral_bWatchdogError:= DiagsRetain.DG_NX5000_3_tGeneral_bWatchdogError OR DG_NX5000_3.tGeneral.bWatchdogError ;
	DiagsRetain.DG_NX5000_3_tNX5000_bNX5000NoCfg:= DiagsRetain.DG_NX5000_3_tNX5000_bNX5000NoCfg OR DG_NX5000_3.tNX5000.bNX5000NoCfg ;
	DiagsRetain.DG_NX5000_3_tNX5000_bStsEthLink:= DiagsRetain.DG_NX5000_3_tNX5000_bStsEthLink OR DG_NX5000_3.tNX5000.bStsEthLink ;	
	
// DG_MODBUS_Master_1
	DiagsRetain.DG_MODBUS_Master_1_tDiag_bConfigFailure:= DiagsRetain.DG_MODBUS_Master_1_tDiag_bConfigFailure OR DG_MODBUS_Master_1.tDiag.bConfigFailure ;
	DiagsRetain.DG_MODBUS_Master_1_tDiag_bModuleFailure:= DiagsRetain.DG_MODBUS_Master_1_tDiag_bModuleFailure OR DG_MODBUS_Master_1.tDiag.bModuleFailure ;
	DiagsRetain.DG_MODBUS_Master_1_tDiag_bRXFailure:= DiagsRetain.DG_MODBUS_Master_1_tDiag_bRXFailure OR DG_MODBUS_Master_1.tDiag.bRXFailure ;
	DiagsRetain.DG_MODBUS_Master_1_tDiag_bTXFailure:= DiagsRetain.DG_MODBUS_Master_1_tDiag_bTXFailure OR DG_MODBUS_Master_1.tDiag.bTXFailure ;
	
// DG_MODBUS_Slave_1
	DiagsRetain.DG_MODBUS_Slave_1_tDiag_bConfigFailure:= DiagsRetain.DG_MODBUS_Slave_1_tDiag_bConfigFailure OR DG_MODBUS_Slave_1.tDiag.bConfigFailure ;
	DiagsRetain.DG_MODBUS_Slave_1_tDiag_bModuleFailure:= DiagsRetain.DG_MODBUS_Slave_1_tDiag_bModuleFailure OR DG_MODBUS_Slave_1.tDiag.bModuleFailure ;
	DiagsRetain.DG_MODBUS_Slave_1_tDiag_bRXFailure:= DiagsRetain.DG_MODBUS_Slave_1_tDiag_bRXFailure OR DG_MODBUS_Slave_1.tDiag.bRXFailure ;
	DiagsRetain.DG_MODBUS_Slave_1_tDiag_bTXFailure:= DiagsRetain.DG_MODBUS_Slave_1_tDiag_bTXFailure OR DG_MODBUS_Slave_1.tDiag.bTXFailure ;
	
// DG_MODBUS_Client_2
	DiagsRetain.DG_MODBUS_Client_2_tDiag_bConfigFailure:= DiagsRetain.DG_MODBUS_Client_2_tDiag_bConfigFailure OR (DG_MODBUS_Client_2.tDiag.bConfigFailure AND bBoolValue) ;
	DiagsRetain.DG_MODBUS_Client_2_tDiag_bModuleFailure:= DiagsRetain.DG_MODBUS_Client_2_tDiag_bModuleFailure OR (DG_MODBUS_Client_2.tDiag.bModuleFailure AND bBoolValue) ;
	DiagsRetain.DG_MODBUS_Client_2_tDiag_bRXFailure:= DiagsRetain.DG_MODBUS_Client_2_tDiag_bRXFailure OR DG_MODBUS_Client_2.tDiag.bRXFailure ;
	DiagsRetain.DG_MODBUS_Client_2_tDiag_bTXFailure:= DiagsRetain.DG_MODBUS_Client_2_tDiag_bTXFailure OR DG_MODBUS_Client_2.tDiag.bTXFailure ;
	
// DG_MODBUS_Server_2
	DiagsRetain.DG_MODBUS_Server_2_tDiag_bConfigFailure:= DiagsRetain.DG_MODBUS_Server_2_tDiag_bConfigFailure OR (DG_MODBUS_Server_2.tDiag.bConfigFailure AND bBoolValue) ;
	DiagsRetain.DG_MODBUS_Server_2_tDiag_bModuleFailure:= DiagsRetain.DG_MODBUS_Server_2_tDiag_bModuleFailure OR (DG_MODBUS_Server_2.tDiag.bModuleFailure AND bBoolValue) ;
	DiagsRetain.DG_MODBUS_Server_2_tDiag_bRXFailure:= DiagsRetain.DG_MODBUS_Server_2_tDiag_bRXFailure OR DG_MODBUS_Server_2.tDiag.bRXFailure ;
	DiagsRetain.DG_MODBUS_Server_2_tDiag_bTXFailure:= DiagsRetain.DG_MODBUS_Server_2_tDiag_bTXFailure OR DG_MODBUS_Server_2.tDiag.bTXFailure ;
	
// DG_MODBUS_Client_3
	DiagsRetain.DG_MODBUS_Client_3_tDiag_bConfigFailure:= DiagsRetain.DG_MODBUS_Client_3_tDiag_bConfigFailure OR (DG_MODBUS_Client_3.tDiag.bConfigFailure AND bBoolValue) ;
	DiagsRetain.DG_MODBUS_Client_3_tDiag_bModuleFailure:= DiagsRetain.DG_MODBUS_Client_3_tDiag_bModuleFailure OR (DG_MODBUS_Client_3.tDiag.bModuleFailure AND bBoolValue) ;
	DiagsRetain.DG_MODBUS_Client_3_tDiag_bRXFailure:= DiagsRetain.DG_MODBUS_Client_3_tDiag_bRXFailure OR DG_MODBUS_Client_3.tDiag.bRXFailure ;
	DiagsRetain.DG_MODBUS_Client_3_tDiag_bTXFailure:= DiagsRetain.DG_MODBUS_Client_3_tDiag_bTXFailure OR DG_MODBUS_Client_3.tDiag.bTXFailure ;
	
// DG_MODBUS_Server_3
	DiagsRetain.DG_MODBUS_Server_3_tDiag_bConfigFailure:= DiagsRetain.DG_MODBUS_Server_3_tDiag_bConfigFailure OR (DG_MODBUS_Server_3.tDiag.bConfigFailure AND bBoolValue) ;
	DiagsRetain.DG_MODBUS_Server_3_tDiag_bModuleFailure:= DiagsRetain.DG_MODBUS_Server_3_tDiag_bModuleFailure OR (DG_MODBUS_Server_3.tDiag.bModuleFailure AND bBoolValue) ;
	DiagsRetain.DG_MODBUS_Server_3_tDiag_bRXFailure:= DiagsRetain.DG_MODBUS_Server_3_tDiag_bRXFailure OR DG_MODBUS_Server_3.tDiag.bRXFailure ;
	DiagsRetain.DG_MODBUS_Server_3_tDiag_bTXFailure:= DiagsRetain.DG_MODBUS_Server_3_tDiag_bTXFailure OR DG_MODBUS_Server_3.tDiag.bTXFailure ;
	
// DG_MODBUS_Client_4
	DiagsRetain.DG_MODBUS_Client_4_tDiag_bConfigFailure:= DiagsRetain.DG_MODBUS_Client_4_tDiag_bConfigFailure OR (DG_MODBUS_Client_4.tDiag.bConfigFailure AND bBoolValue) ;
	DiagsRetain.DG_MODBUS_Client_4_tDiag_bModuleFailure:= DiagsRetain.DG_MODBUS_Client_4_tDiag_bModuleFailure OR (DG_MODBUS_Client_4.tDiag.bModuleFailure AND bBoolValue) ;
	DiagsRetain.DG_MODBUS_Client_4_tDiag_bRXFailure:= DiagsRetain.DG_MODBUS_Client_4_tDiag_bRXFailure OR DG_MODBUS_Client_4.tDiag.bRXFailure ;
	DiagsRetain.DG_MODBUS_Client_4_tDiag_bTXFailure:= DiagsRetain.DG_MODBUS_Client_4_tDiag_bTXFailure OR DG_MODBUS_Client_4.tDiag.bTXFailure ;
	
// DG_MODBUS_Server_4
	DiagsRetain.DG_MODBUS_Server_4_tDiag_bConfigFailure:= DiagsRetain.DG_MODBUS_Server_4_tDiag_bConfigFailure OR (DG_MODBUS_Server_4.tDiag.bConfigFailure AND bBoolValue) ;
	DiagsRetain.DG_MODBUS_Server_4_tDiag_bModuleFailure:= DiagsRetain.DG_MODBUS_Server_4_tDiag_bModuleFailure OR (DG_MODBUS_Server_4.tDiag.bModuleFailure AND bBoolValue) ;
	DiagsRetain.DG_MODBUS_Server_4_tDiag_bRXFailure:= DiagsRetain.DG_MODBUS_Server_4_tDiag_bRXFailure OR DG_MODBUS_Server_4.tDiag.bRXFailure ;
	DiagsRetain.DG_MODBUS_Server_4_tDiag_bTXFailure:= DiagsRetain.DG_MODBUS_Server_4_tDiag_bTXFailure OR DG_MODBUS_Server_4.tDiag.bTXFailure ;
	
	
//PO1000				
	DiagsRetain.DG_REM05_PO1000_bHardwareFailure	:=	DiagsRetain.DG_REM05_PO1000_bHardwareFailure	OR	DG_REM05_PO1000.bHardwareFailure;
	DiagsRetain.DG_REM05_PO1000_bPowerSupplyFail	:=	DiagsRetain.DG_REM05_PO1000_bPowerSupplyFail	or	DG_REM05_PO1000.bPowerSupplyFail;
					
//PO2020				
	DiagsRetain.DG_REM05_PO2020_bHardwareFailure	:=	DiagsRetain.DG_REM05_PO2020_bHardwareFailure	OR	DG_REM05_PO2020.bHardwareFailure;
	DiagsRetain.DG_REM05_PO2020_bPowerSupplyFail	:=	DiagsRetain.DG_REM05_PO2020_bPowerSupplyFail	or	DG_REM05_PO2020.bPowerSupplyFail;
					
//PO9100				
	DiagsRetain.DG_REM05_PO9100_bReserved00	:=	DiagsRetain.DG_REM05_PO9100_bReserved00	OR	DG_REM05_PO9100.bReserved00;
					
//PO1212				
	DiagsRetain.DG_REM10_PO1212_bFuseOpen	:=	DiagsRetain.DG_REM10_PO1212_bFuseOpen	OR	DG_REM10_PO1212.bFuseOpen;
	DiagsRetain.DG_REM10_PO1212_bHardwareFailure	:=	DiagsRetain.DG_REM10_PO1212_bHardwareFailure	or	DG_REM10_PO1212.bHardwareFailure;
	DiagsRetain.DG_REM10_PO1212_bNoParametrizedModule	:=	DiagsRetain.DG_REM10_PO1212_bNoParametrizedModule	or	DG_REM10_PO1212.bNoParametrizedModule;
	DiagsRetain.DG_REM10_PO1212_bOverTemp	:=	DiagsRetain.DG_REM10_PO1212_bOverTemp	or	DG_REM10_PO1212.bOverTemp;
	DiagsRetain.DG_REM10_PO1212_aCh0_bOpenSensor	:=	DiagsRetain.DG_REM10_PO1212_aCh0_bOpenSensor	or	DG_REM10_PO1212.aCh[0].bOpenSensor;
	DiagsRetain.DG_REM10_PO1212_aCh0_bOverRange	:=	DiagsRetain.DG_REM10_PO1212_aCh0_bOverRange	or	DG_REM10_PO1212.aCh[0].bOverRange;
	DiagsRetain.DG_REM10_PO1212_aCh0_bSensorShortCircuit	:=	DiagsRetain.DG_REM10_PO1212_aCh0_bSensorShortCircuit	or	DG_REM10_PO1212.aCh[0].bSensorShortCircuit;
	DiagsRetain.DG_REM10_PO1212_aCh0_bWrongParameters	:=	DiagsRetain.DG_REM10_PO1212_aCh0_bWrongParameters	or	DG_REM10_PO1212.aCh[0].bWrongParameters;
	DiagsRetain.DG_REM10_PO1212_aCh1_bOpenSensor	:=	DiagsRetain.DG_REM10_PO1212_aCh1_bOpenSensor	or	DG_REM10_PO1212.aCh[1].bOpenSensor;
	DiagsRetain.DG_REM10_PO1212_aCh1_bOverRange	:=	DiagsRetain.DG_REM10_PO1212_aCh1_bOverRange	or	DG_REM10_PO1212.aCh[1].bOverRange;
	DiagsRetain.DG_REM10_PO1212_aCh1_bSensorShortCircuit	:=	DiagsRetain.DG_REM10_PO1212_aCh1_bSensorShortCircuit	or	DG_REM10_PO1212.aCh[1].bSensorShortCircuit;
	DiagsRetain.DG_REM10_PO1212_aCh1_bWrongParameters	:=	DiagsRetain.DG_REM10_PO1212_aCh1_bWrongParameters	or	DG_REM10_PO1212.aCh[1].bWrongParameters;
	DiagsRetain.DG_REM10_PO1212_aCh2_bOpenSensor	:=	DiagsRetain.DG_REM10_PO1212_aCh2_bOpenSensor	or	DG_REM10_PO1212.aCh[2].bOpenSensor;
	DiagsRetain.DG_REM10_PO1212_aCh2_bOverRange	:=	DiagsRetain.DG_REM10_PO1212_aCh2_bOverRange	or	DG_REM10_PO1212.aCh[2].bOverRange;
	DiagsRetain.DG_REM10_PO1212_aCh2_bSensorShortCircuit	:=	DiagsRetain.DG_REM10_PO1212_aCh2_bSensorShortCircuit	or	DG_REM10_PO1212.aCh[2].bSensorShortCircuit;
	DiagsRetain.DG_REM10_PO1212_aCh2_bWrongParameters	:=	DiagsRetain.DG_REM10_PO1212_aCh2_bWrongParameters	or	DG_REM10_PO1212.aCh[2].bWrongParameters;
	DiagsRetain.DG_REM10_PO1212_aCh3_bOpenSensor	:=	DiagsRetain.DG_REM10_PO1212_aCh3_bOpenSensor	or	DG_REM10_PO1212.aCh[3].bOpenSensor;
	DiagsRetain.DG_REM10_PO1212_aCh3_bOverRange	:=	DiagsRetain.DG_REM10_PO1212_aCh3_bOverRange	or	DG_REM10_PO1212.aCh[3].bOverRange;
	DiagsRetain.DG_REM10_PO1212_aCh3_bSensorShortCircuit	:=	DiagsRetain.DG_REM10_PO1212_aCh3_bSensorShortCircuit	or	DG_REM10_PO1212.aCh[3].bSensorShortCircuit;
	DiagsRetain.DG_REM10_PO1212_aCh3_bWrongParameters	:=	DiagsRetain.DG_REM10_PO1212_aCh3_bWrongParameters	or	DG_REM10_PO1212.aCh[3].bWrongParameters;
	DiagsRetain.DG_REM10_PO1212_aCh4_bOpenSensor	:=	DiagsRetain.DG_REM10_PO1212_aCh4_bOpenSensor	or	DG_REM10_PO1212.aCh[4].bOpenSensor;
	DiagsRetain.DG_REM10_PO1212_aCh4_bOverRange	:=	DiagsRetain.DG_REM10_PO1212_aCh4_bOverRange	or	DG_REM10_PO1212.aCh[4].bOverRange;
	DiagsRetain.DG_REM10_PO1212_aCh4_bSensorShortCircuit	:=	DiagsRetain.DG_REM10_PO1212_aCh4_bSensorShortCircuit	or	DG_REM10_PO1212.aCh[4].bSensorShortCircuit;
	DiagsRetain.DG_REM10_PO1212_aCh4_bWrongParameters	:=	DiagsRetain.DG_REM10_PO1212_aCh4_bWrongParameters	or	DG_REM10_PO1212.aCh[4].bWrongParameters;
	DiagsRetain.DG_REM10_PO1212_aCh5_bOpenSensor	:=	DiagsRetain.DG_REM10_PO1212_aCh5_bOpenSensor	or	DG_REM10_PO1212.aCh[5].bOpenSensor;
	DiagsRetain.DG_REM10_PO1212_aCh5_bOverRange	:=	DiagsRetain.DG_REM10_PO1212_aCh5_bOverRange	or	DG_REM10_PO1212.aCh[5].bOverRange;
	DiagsRetain.DG_REM10_PO1212_aCh5_bSensorShortCircuit	:=	DiagsRetain.DG_REM10_PO1212_aCh5_bSensorShortCircuit	or	DG_REM10_PO1212.aCh[5].bSensorShortCircuit;
	DiagsRetain.DG_REM10_PO1212_aCh5_bWrongParameters	:=	DiagsRetain.DG_REM10_PO1212_aCh5_bWrongParameters	or	DG_REM10_PO1212.aCh[5].bWrongParameters;
	DiagsRetain.DG_REM10_PO1212_aCh6_bOpenSensor	:=	DiagsRetain.DG_REM10_PO1212_aCh6_bOpenSensor	or	DG_REM10_PO1212.aCh[6].bOpenSensor;
	DiagsRetain.DG_REM10_PO1212_aCh6_bOverRange	:=	DiagsRetain.DG_REM10_PO1212_aCh6_bOverRange	or	DG_REM10_PO1212.aCh[6].bOverRange;
	DiagsRetain.DG_REM10_PO1212_aCh6_bSensorShortCircuit	:=	DiagsRetain.DG_REM10_PO1212_aCh6_bSensorShortCircuit	or	DG_REM10_PO1212.aCh[6].bSensorShortCircuit;
	DiagsRetain.DG_REM10_PO1212_aCh6_bWrongParameters	:=	DiagsRetain.DG_REM10_PO1212_aCh6_bWrongParameters	or	DG_REM10_PO1212.aCh[6].bWrongParameters;
	DiagsRetain.DG_REM10_PO1212_aCh7_bOpenSensor	:=	DiagsRetain.DG_REM10_PO1212_aCh7_bOpenSensor	or	DG_REM10_PO1212.aCh[7].bOpenSensor;
	DiagsRetain.DG_REM10_PO1212_aCh7_bOverRange	:=	DiagsRetain.DG_REM10_PO1212_aCh7_bOverRange	or	DG_REM10_PO1212.aCh[7].bOverRange;
	DiagsRetain.DG_REM10_PO1212_aCh7_bSensorShortCircuit	:=	DiagsRetain.DG_REM10_PO1212_aCh7_bSensorShortCircuit	or	DG_REM10_PO1212.aCh[7].bSensorShortCircuit;
	DiagsRetain.DG_REM10_PO1212_aCh7_bWrongParameters	:=	DiagsRetain.DG_REM10_PO1212_aCh7_bWrongParameters	or	DG_REM10_PO1212.aCh[7].bWrongParameters;
					
//PO2132				
	DiagsRetain.DG_REM10_PO2132_bNoParametrizedModule	:=	DiagsRetain.DG_REM10_PO2132_bNoParametrizedModule	OR	DG_REM10_PO2132.bNoParametrizedModule;
	DiagsRetain.DG_REM10_PO2132_bPowerSupplyFail	:=	DiagsRetain.DG_REM10_PO2132_bPowerSupplyFail	or	DG_REM10_PO2132.bPowerSupplyFail;
	DiagsRetain.DG_REM10_PO2132_aCh0_bOpenSensor	:=	DiagsRetain.DG_REM10_PO2132_aCh0_bOpenSensor	or	DG_REM10_PO2132.aCh[0].bOpenSensor;
	DiagsRetain.DG_REM10_PO2132_aCh0_bWrongParameters	:=	DiagsRetain.DG_REM10_PO2132_aCh0_bWrongParameters	or	DG_REM10_PO2132.aCh[0].bWrongParameters;
	DiagsRetain.DG_REM10_PO2132_aCh1_bOpenSensor	:=	DiagsRetain.DG_REM10_PO2132_aCh1_bOpenSensor	or	DG_REM10_PO2132.aCh[1].bOpenSensor;
	DiagsRetain.DG_REM10_PO2132_aCh1_bWrongParameters	:=	DiagsRetain.DG_REM10_PO2132_aCh1_bWrongParameters	or	DG_REM10_PO2132.aCh[1].bWrongParameters;
	DiagsRetain.DG_REM10_PO2132_aCh2_bOpenSensor	:=	DiagsRetain.DG_REM10_PO2132_aCh2_bOpenSensor	or	DG_REM10_PO2132.aCh[2].bOpenSensor;
	DiagsRetain.DG_REM10_PO2132_aCh2_bWrongParameters	:=	DiagsRetain.DG_REM10_PO2132_aCh2_bWrongParameters	or	DG_REM10_PO2132.aCh[2].bWrongParameters;
	DiagsRetain.DG_REM10_PO2132_aCh3_bOpenSensor	:=	DiagsRetain.DG_REM10_PO2132_aCh3_bOpenSensor	or	DG_REM10_PO2132.aCh[3].bOpenSensor;
	DiagsRetain.DG_REM10_PO2132_aCh3_bWrongParameters	:=	DiagsRetain.DG_REM10_PO2132_aCh3_bWrongParameters	or	DG_REM10_PO2132.aCh[3].bWrongParameters;

					
//PO9100				
	DiagsRetain.DG_REM10_PO9100_bReserved00	:=	DiagsRetain.DG_REM10_PO9100_bReserved00	OR	DG_REM10_PO9100.bReserved00;
					
//PO1000				
	DiagsRetain.DG_REM04_PO1000_bHardwareFailure	:=	DiagsRetain.DG_REM04_PO1000_bHardwareFailure	OR	DG_REM04_PO1000.bHardwareFailure;
	DiagsRetain.DG_REM04_PO1000_bPowerSupplyFail	:=	DiagsRetain.DG_REM04_PO1000_bPowerSupplyFail	or	DG_REM04_PO1000.bPowerSupplyFail;

	
	// Se este for o PLCA e ele está no estado ativo...
IF DG_NX4010.tRedundancy.RedDgnLoc.sGeneral_Diag.eRedState = REDUNDANCY_STATE.ACTIVE AND 
   DG_NX4010.tRedundancy.RedDgnLoc.sGeneral_Diag.ePLC_ID = CLUCONF_ID.PLC_A THEN
	IF 		
	// NX3030
		DiagsRetain.DG_NX3030_tSummarized_bAbsentModules OR
		DiagsRetain.DG_NX3030_tSummarized_bAbsentRacks OR
		DiagsRetain.DG_NX3030_tSummarized_bCOM1ConfigError OR
		DiagsRetain.DG_NX3030_tSummarized_bCOM2ConfigError OR
		DiagsRetain.DG_NX3030_tSummarized_bConfigMismatch OR
		DiagsRetain.DG_NX3030_tSummarized_bDuplicatedRacks OR
		DiagsRetain.DG_NX3030_tSummarized_bDuplicatedSlots OR
		DiagsRetain.DG_NX3030_tSummarized_bHardwareFailure OR
		DiagsRetain.DG_NX3030_tSummarized_bInvalidDateTime OR
		DiagsRetain.DG_NX3030_tSummarized_bInvalidRacks OR
		DiagsRetain.DG_NX3030_tSummarized_bMemoryCardError OR
		DiagsRetain.DG_NX3030_tSummarized_bModuleFatalError OR
		DiagsRetain.DG_NX3030_tSummarized_bModuleParameterError OR
		DiagsRetain.DG_NX3030_tSummarized_bModulesWithDiagnostic OR
		DiagsRetain.DG_NX3030_tSummarized_bNET1ConfigError OR
		DiagsRetain.DG_NX3030_tSummarized_bNET2ConfigError OR
		DiagsRetain.DG_NX3030_tSummarized_bNonDeclaredModules OR
		DiagsRetain.DG_NX3030_tSummarized_bNonDeclaredRacks OR
		DiagsRetain.DG_NX3030_tSummarized_bOTDSwitchError OR
		DiagsRetain.DG_NX3030_tSummarized_bRuntimeReset OR
		DiagsRetain.DG_NX3030_tSummarized_bSoftwareException OR
		DiagsRetain.DG_NX3030_tSummarized_bSwappedModules OR
		DiagsRetain.DG_NX3030_tSummarized_bWHSBBusError OR
		DiagsRetain.DG_NX3030_tDetailed_MemoryCard_byMounted OR
		DiagsRetain.DG_NX3030_tDetailed_Ethernet_NET1_bLinkDown OR
		DiagsRetain.DG_NX3030_tDetailed_Ethernet_NET2_bLinkDown OR 
		DiagsRetain.DG_NX3030_tDetailed_Application_byCPUState OR
		DiagsRetain.DG_NX3030_tDetailed_ApplicationInfo_dwApplicationCRC OR
		DiagsRetain.DG_NX3030_tDetailed_Ethernet_NET1_abyMAC_0 OR
		DiagsRetain.DG_NX3030_tDetailed_Ethernet_NET1_abyMAC_1 OR
		DiagsRetain.DG_NX3030_tDetailed_Ethernet_NET1_abyMAC_2 OR
		DiagsRetain.DG_NX3030_tDetailed_Ethernet_NET1_abyMAC_3 OR
		DiagsRetain.DG_NX3030_tDetailed_Ethernet_NET1_abyMAC_4 OR
		DiagsRetain.DG_NX3030_tDetailed_Ethernet_NET1_abyMAC_5 OR
		DiagsRetain.DG_NX3030_tDetailed_Ethernet_NET2_abyMAC_0 OR
		DiagsRetain.DG_NX3030_tDetailed_Ethernet_NET2_abyMAC_1 OR
		DiagsRetain.DG_NX3030_tDetailed_Ethernet_NET2_abyMAC_2 OR
		DiagsRetain.DG_NX3030_tDetailed_Ethernet_NET2_abyMAC_3 OR
		DiagsRetain.DG_NX3030_tDetailed_Ethernet_NET2_abyMAC_4 OR
		DiagsRetain.DG_NX3030_tDetailed_Ethernet_NET2_abyMAC_5 OR
		DiagsRetain.DG_NX3030_tDetailed_Ethernet_NETx_abyIP_0 OR
		DiagsRetain.DG_NX3030_tDetailed_Ethernet_NETx_abyIP_1 OR
		DiagsRetain.DG_NX3030_tDetailed_Ethernet_NETx_abyIP_2 OR
		DiagsRetain.DG_NX3030_tDetailed_Ethernet_NETx_abyIP_3 OR
		DiagsRetain.DG_NX3030_tDetailed_Ethernet_NETx_abyMask_0 OR
		DiagsRetain.DG_NX3030_tDetailed_Ethernet_NETx_abyMask_1 OR
		DiagsRetain.DG_NX3030_tDetailed_Ethernet_NETx_abyMask_2 OR
		DiagsRetain.DG_NX3030_tDetailed_Ethernet_NETx_abyMask_3 OR
		DiagsRetain.DG_NX3030_tDetailed_Ethernet_NETx_abyGateway_0 OR
		DiagsRetain.DG_NX3030_tDetailed_Ethernet_NETx_abyGateway_1 OR
		DiagsRetain.DG_NX3030_tDetailed_Ethernet_NETx_abyGateway_2 OR
		DiagsRetain.DG_NX3030_tDetailed_Ethernet_NETx_abyGateway_3 OR
		DiagsRetain.DG_NX3030_tDetailed_SNTP_bServiceEnabled OR
		DiagsRetain.DG_NX3030_tDetailed_Target_abyAuxprocVersion OR
		DiagsRetain.DG_NX3030_tDetailed_Target_abyBootloaderVersion OR
		DiagsRetain.DG_NX3030_tDetailed_Target_abyCPUVersion OR
		DiagsRetain.DG_NX3030_tDetailed_Target_dwCPUModel OR
		DiagsRetain.DG_NX3030_tDetailed_Thermometer_diTemperature THEN
    bDiag_Error_NX3030:= TRUE;
	ELSE
		bDiag_Error_NX3030:= FALSE;	
	END_IF
	
	IF	
	// NX4010
		DiagsRetain.DG_NX4010_tGeneral_bActiveDiagnostics OR
		DiagsRetain.DG_NX4010_tGeneral_bBusCommunicationError OR
		DiagsRetain.DG_NX4010_tGeneral_bConfigMismatch OR
		DiagsRetain.DG_NX4010_tGeneral_bFatalError OR
		DiagsRetain.DG_NX4010_tGeneral_bNET1LinkDown OR
		DiagsRetain.DG_NX4010_tGeneral_bNET2LinkDown OR
		DiagsRetain.DG_NX4010_tGeneral_bOTDSwitchError OR
		DiagsRetain.DG_NX4010_tGeneral_bWatchdogError OR
		DiagsRetain.DG_NX4010_tRedundancy_RedDgnLoc_sGeneral_Diag_bApplicationIncompatible OR
		DiagsRetain.DG_NX4010_tRedundancy_RedDgnLoc_sGeneral_Diag_bApplicationProjectDiff OR
		DiagsRetain.DG_NX4010_tRedundancy_RedDgnLoc_sGeneral_Diag_bConfigError OR
		DiagsRetain.DG_NX4010_tRedundancy_RedDgnLoc_sGeneral_Diag_bExchangeSync OR
		DiagsRetain.DG_NX4010_tRedundancy_RedDgnLoc_sGeneral_Diag_bFailedPBUS1A OR
		DiagsRetain.DG_NX4010_tRedundancy_RedDgnLoc_sGeneral_Diag_bFailedPBUS1B OR
		DiagsRetain.DG_NX4010_tRedundancy_RedDgnLoc_sGeneral_Diag_bFailedPBUS2A OR
		DiagsRetain.DG_NX4010_tRedundancy_RedDgnLoc_sGeneral_Diag_bFailedPBUS2B OR
		DiagsRetain.DG_NX4010_tRedundancy_RedDgnLoc_sGeneral_Diag_bFailedRED OR
		DiagsRetain.DG_NX4010_tRedundancy_RedDgnLoc_sGeneral_Diag_bFailureProfibus_1 OR
		DiagsRetain.DG_NX4010_tRedundancy_RedDgnLoc_sGeneral_Diag_bFailureProfibus_2 OR
		DiagsRetain.DG_NX4010_tRedundancy_RedDgnLoc_sGeneral_Diag_bIncompatibleFirmware OR
		DiagsRetain.DG_NX4010_tRedundancy_RedDgnLoc_sGeneral_Diag_bProfibusVitalFailureAll OR
		DiagsRetain.DG_NX4010_tRedundancy_RedDgnLoc_sGeneral_Diag_bProfibusVitalFailureAny OR
		DiagsRetain.DG_NX4010_tRedundancy_RedDgnLoc_sGeneral_Diag_bProjectArchiveDiff OR
		DiagsRetain.DG_NX4010_tRedundancy_RedDgnLoc_sGeneral_Diag_bProjectSyncDisable OR
		DiagsRetain.DG_NX4010_tRedundancy_RedDgnLoc_sGeneral_Diag_bRedDataSync OR
		DiagsRetain.DG_NX4010_tRedundancy_RedDgnLoc_sGeneral_Diag_bRedForceSync OR
		DiagsRetain.DG_NX4010_tRedundancy_RedDgnLoc_sGeneral_Diag_bRedPanelTestMode OR
		DiagsRetain.DG_NX4010_tRedundancy_RedDgnLoc_sGeneral_Diag_bTemporaryBufferTooSmall OR
		DiagsRetain.DG_NX4010_tRedundancy_RedDgnLoc_sGeneral_Diag_bTooManyRedAreas OR
		DiagsRetain.DG_NX4010_tRedundancy_RedDgnLoc_sGeneral_Diag_dwArchiveCRC OR  // Demanda 19831
		DiagsRetain.DG_NX4010_tRedundancy_RedDgnLoc_sGeneral_Diag_dwApplicationCRC THEN
    	bDiag_Error_NX4010:= TRUE;
	ELSE
		bDiag_Error_NX4010:= FALSE;	
	END_IF
	
	IF		
	// NX5001_1
		DiagsRetain.DG_NX5001_1_tGeneral_bActiveDiagnostics OR
		DiagsRetain.DG_NX5001_1_tGeneral_bBusCommunicationError OR
		DiagsRetain.DG_NX5001_1_tGeneral_bConfigMismatch OR
		DiagsRetain.DG_NX5001_1_tGeneral_bFatalError OR
		DiagsRetain.DG_NX5001_1_tGeneral_bNX5001NoCfg OR
		DiagsRetain.DG_NX5001_1_tGeneral_bOTDSwitchError OR
		DiagsRetain.DG_NX5001_1_tGeneral_bPbusCommFail OR
		DiagsRetain.DG_NX5001_1_tGeneral_bSlaveNotConfigured OR
		DiagsRetain.DG_NX5001_1_tGeneral_bSlaveNotPresent OR
		DiagsRetain.DG_NX5001_1_tGeneral_bSlaveWithDiagnostic OR
		DiagsRetain.DG_NX5001_1_tGeneral_bStsEnableInterface OR
	//	DiagsRetain.DG_NX5001_1_tGeneral_bStsMstRedundEnable OR   Demanda 17571
		DiagsRetain.DG_NX5001_1_tGeneral_bWatchdogError THEN
    	bDiag_Error_NX5001_1:= TRUE;
	ELSE
		bDiag_Error_NX5001_1:= FALSE;	
	END_IF
	
	IF
	// NX5001_2
		DiagsRetain.DG_NX5001_2_tGeneral_bActiveDiagnostics OR
		DiagsRetain.DG_NX5001_2_tGeneral_bBusCommunicationError OR
		DiagsRetain.DG_NX5001_2_tGeneral_bConfigMismatch OR
		DiagsRetain.DG_NX5001_2_tGeneral_bFatalError OR
		DiagsRetain.DG_NX5001_2_tGeneral_bNX5001NoCfg OR
		DiagsRetain.DG_NX5001_2_tGeneral_bOTDSwitchError OR
		DiagsRetain.DG_NX5001_2_tGeneral_bPbusCommFail OR
		DiagsRetain.DG_NX5001_2_tGeneral_bSlaveNotConfigured OR
		DiagsRetain.DG_NX5001_2_tGeneral_bSlaveNotPresent OR
		DiagsRetain.DG_NX5001_2_tGeneral_bSlaveWithDiagnostic OR
		DiagsRetain.DG_NX5001_2_tGeneral_bStsEnableInterface OR
	//	DiagsRetain.DG_NX5001_2_tGeneral_bStsMstRedundEnable OR   Demanda 17571
		DiagsRetain.DG_NX5001_2_tGeneral_bWatchdogError THEN
   	 	bDiag_Error_NX5001_2:= TRUE;
	ELSE
		bDiag_Error_NX5001_2:= FALSE;	
	END_IF
	
	IF
	// NX5001_3
		DiagsRetain.DG_NX5001_3_tGeneral_bActiveDiagnostics OR
		DiagsRetain.DG_NX5001_3_tGeneral_bBusCommunicationError OR
		DiagsRetain.DG_NX5001_3_tGeneral_bConfigMismatch OR
		DiagsRetain.DG_NX5001_3_tGeneral_bFatalError OR
		DiagsRetain.DG_NX5001_3_tGeneral_bNX5001NoCfg OR
		DiagsRetain.DG_NX5001_3_tGeneral_bOTDSwitchError OR
		DiagsRetain.DG_NX5001_3_tGeneral_bPbusCommFail OR
		DiagsRetain.DG_NX5001_3_tGeneral_bSlaveNotConfigured OR
		DiagsRetain.DG_NX5001_3_tGeneral_bSlaveNotPresent OR
		DiagsRetain.DG_NX5001_3_tGeneral_bSlaveWithDiagnostic OR
		DiagsRetain.DG_NX5001_3_tGeneral_bStsEnableInterface OR
	//	DiagsRetain.DG_NX5001_3_tGeneral_bStsMstRedundEnable OR   Demanda 17571
		DiagsRetain.DG_NX5001_3_tGeneral_bWatchdogError THEN
  	 	bDiag_Error_NX5001_3:= TRUE;
	ELSE
		bDiag_Error_NX5001_3:= FALSE;	
	END_IF
	
	IF
	// NX5000_1	
		DiagsRetain.DG_NX5000_1_tGeneral_bActiveDiagnostics OR
		DiagsRetain.DG_NX5000_1_tGeneral_bBusCommunicationError OR
		DiagsRetain.DG_NX5000_1_tGeneral_bConfigMismatch OR
		DiagsRetain.DG_NX5000_1_tGeneral_bFatalError OR
		DiagsRetain.DG_NX5000_1_tGeneral_bOTDSwitchError OR
		DiagsRetain.DG_NX5000_1_tGeneral_bWatchdogError OR
		DiagsRetain.DG_NX5000_1_tNX5000_bNX5000NoCfg OR
		DiagsRetain.DG_NX5000_1_tNX5000_bStsEthLink THEN
    	bDiag_Error_NX5000_1:= TRUE;
	ELSE
		bDiag_Error_NX5000_1:= FALSE;	
	END_IF
	
	IF
	// NX5000_2	
		DiagsRetain.DG_NX5000_2_tGeneral_bActiveDiagnostics OR
		DiagsRetain.DG_NX5000_2_tGeneral_bBusCommunicationError OR
		DiagsRetain.DG_NX5000_2_tGeneral_bConfigMismatch OR
		DiagsRetain.DG_NX5000_2_tGeneral_bFatalError OR
		DiagsRetain.DG_NX5000_2_tGeneral_bOTDSwitchError OR
		DiagsRetain.DG_NX5000_2_tGeneral_bWatchdogError OR
		DiagsRetain.DG_NX5000_2_tNX5000_bNX5000NoCfg OR
		DiagsRetain.DG_NX5000_2_tNX5000_bStsEthLink THEN
    	bDiag_Error_NX5000_2:= TRUE;
	ELSE
		bDiag_Error_NX5000_2:= FALSE;	
	END_IF
	
	IF
	// NX5000_3	
		DiagsRetain.DG_NX5000_3_tGeneral_bActiveDiagnostics OR
		DiagsRetain.DG_NX5000_3_tGeneral_bBusCommunicationError OR
		DiagsRetain.DG_NX5000_3_tGeneral_bConfigMismatch OR
		DiagsRetain.DG_NX5000_3_tGeneral_bFatalError OR
		DiagsRetain.DG_NX5000_3_tGeneral_bOTDSwitchError OR
		DiagsRetain.DG_NX5000_3_tGeneral_bWatchdogError OR
		DiagsRetain.DG_NX5000_3_tNX5000_bNX5000NoCfg OR
		DiagsRetain.DG_NX5000_3_tNX5000_bStsEthLink THEN
    	bDiag_Error_NX5000_3:= TRUE;
	ELSE
		bDiag_Error_NX5000_3:= FALSE;	
	END_IF
	
	IF
	// DiagsRetain.DG_MODBUS_Master_1
		DiagsRetain.DG_MODBUS_Master_1_tDiag_bConfigFailure OR
		DiagsRetain.DG_MODBUS_Master_1_tDiag_bModuleFailure OR
		DiagsRetain.DG_MODBUS_Master_1_tDiag_bRXFailure OR
		DiagsRetain.DG_MODBUS_Master_1_tDiag_bTXFailure THEN
   	 	bDiag_Error_MODBUS_Master_1:= TRUE;
	ELSE
		bDiag_Error_MODBUS_Master_1:= FALSE;	
	END_IF
	
	IF
	// MODBUS_Slave_1	
		DiagsRetain.DG_MODBUS_Slave_1_tDiag_bConfigFailure OR
		DiagsRetain.DG_MODBUS_Slave_1_tDiag_bModuleFailure OR
		DiagsRetain.DG_MODBUS_Slave_1_tDiag_bRXFailure OR
		DiagsRetain.DG_MODBUS_Slave_1_tDiag_bTXFailure THEN
   		bDiag_Error_MODBUS_Slave_1:= TRUE;
	ELSE
		bDiag_Error_MODBUS_Slave_1:= FALSE;	
	END_IF
	
	IF
	// MODBUS_Client_2
		DiagsRetain.DG_MODBUS_Client_2_tDiag_bConfigFailure OR
//		DiagsRetain.DG_MODBUS_Client_2_tDiag_bModuleFailure OR 	// Demanda 13816
		DiagsRetain.DG_MODBUS_Client_2_tDiag_bRXFailure OR
		DiagsRetain.DG_MODBUS_Client_2_tDiag_bTXFailure THEN
    	bDiag_Error_MODBUS_Client_2:= TRUE;
	ELSE
		bDiag_Error_MODBUS_Client_2:= FALSE;	
	END_IF
	
	IF
	// MODBUS_Server_2
		DiagsRetain.DG_MODBUS_Server_2_tDiag_bConfigFailure OR
		DiagsRetain.DG_MODBUS_Server_2_tDiag_bModuleFailure OR
		DiagsRetain.DG_MODBUS_Server_2_tDiag_bRXFailure OR
		DiagsRetain.DG_MODBUS_Server_2_tDiag_bTXFailure THEN
    	bDiag_Error_MODBUS_Server_2:= TRUE;
	ELSE
		bDiag_Error_MODBUS_Server_2:= FALSE;	
	END_IF
	
	IF
	// MODBUS_Client_3
		DiagsRetain.DG_MODBUS_Client_3_tDiag_bConfigFailure OR
		DiagsRetain.DG_MODBUS_Client_3_tDiag_bModuleFailure OR
		DiagsRetain.DG_MODBUS_Client_3_tDiag_bRXFailure OR
		DiagsRetain.DG_MODBUS_Client_3_tDiag_bTXFailure THEN
    	bDiag_Error_MODBUS_Client_3:= TRUE;
	ELSE
		bDiag_Error_MODBUS_Client_3:= FALSE;	
	END_IF
	
	IF
	// MODBUS_Server_3
		DiagsRetain.DG_MODBUS_Server_3_tDiag_bConfigFailure OR
//		DiagsRetain.DG_MODBUS_Server_3_tDiag_bModuleFailure OR  	// Demanda 13816
		DiagsRetain.DG_MODBUS_Server_3_tDiag_bRXFailure OR
		DiagsRetain.DG_MODBUS_Server_3_tDiag_bTXFailure THEN
    	bDiag_Error_MODBUS_Server_3:= TRUE;
	ELSE
		bDiag_Error_MODBUS_Server_3:= FALSE;	
	END_IF
	
	IF
	// MODBUS_Client_4
		DiagsRetain.DG_MODBUS_Client_4_tDiag_bConfigFailure OR
		DiagsRetain.DG_MODBUS_Client_4_tDiag_bModuleFailure OR
		DiagsRetain.DG_MODBUS_Client_4_tDiag_bRXFailure OR
		DiagsRetain.DG_MODBUS_Client_4_tDiag_bTXFailure THEN
    	bDiag_Error_MODBUS_Client_4:= TRUE;
	ELSE
		bDiag_Error_MODBUS_Client_4:= FALSE;	
	END_IF
	
	IF
	// MODBUS_Server_4	
		DiagsRetain.DG_MODBUS_Server_4_tDiag_bConfigFailure OR
//		DiagsRetain.DG_MODBUS_Server_4_tDiag_bModuleFailure OR  	// Demanda 13816
		DiagsRetain.DG_MODBUS_Server_4_tDiag_bRXFailure OR
		DiagsRetain.DG_MODBUS_Server_4_tDiag_bTXFailure THEN
    	bDiag_Error_MODBUS_Server_4:= TRUE;
	ELSE
		bDiag_Error_MODBUS_Server_4:= FALSE;	
	END_IF
	
	IF		
		//PO1000
		DiagsRetain.DG_REM05_PO1000_bHardwareFailure OR
		DiagsRetain.DG_REM05_PO1000_bPowerSupplyFail THEN
	   	bDiag_Error_PO1000_REM05:= TRUE;
	ELSE
		bDiag_Error_PO1000_REM05:= FALSE;	
	END_IF
	
	IF		
		//PO2020
		DiagsRetain.DG_REM05_PO2020_bHardwareFailure OR
		DiagsRetain.DG_REM05_PO2020_bPowerSupplyFail THEN
		bDiag_Error_PO2020_REM05:= TRUE;
	ELSE
		bDiag_Error_PO2020_REM05:= FALSE;	
	END_IF

	IF		
		//PO9100	
		DiagsRetain.DG_REM05_PO9100_bReserved00 THEN
		bDiag_Error_PO9100_REM05:= TRUE;
	ELSE
		bDiag_Error_PO9100_REM05:= FALSE;	
	END_IF	
	
	IF		
	//PO1212
	DiagsRetain.DG_REM10_PO1212_bFuseOpen OR
	DiagsRetain.DG_REM10_PO1212_bHardwareFailure OR
	DiagsRetain.DG_REM10_PO1212_bNoParametrizedModule OR
	DiagsRetain.DG_REM10_PO1212_bOverTemp OR
	DiagsRetain.DG_REM10_PO1212_aCh0_bOpenSensor OR
	DiagsRetain.DG_REM10_PO1212_aCh0_bOverRange OR
	DiagsRetain.DG_REM10_PO1212_aCh0_bSensorShortCircuit OR
	DiagsRetain.DG_REM10_PO1212_aCh0_bWrongParameters OR
	DiagsRetain.DG_REM10_PO1212_aCh1_bOpenSensor OR
	DiagsRetain.DG_REM10_PO1212_aCh1_bOverRange OR
	DiagsRetain.DG_REM10_PO1212_aCh1_bSensorShortCircuit OR
	DiagsRetain.DG_REM10_PO1212_aCh1_bWrongParameters OR
	DiagsRetain.DG_REM10_PO1212_aCh2_bOpenSensor OR
	DiagsRetain.DG_REM10_PO1212_aCh2_bOverRange OR
	DiagsRetain.DG_REM10_PO1212_aCh2_bSensorShortCircuit OR
	DiagsRetain.DG_REM10_PO1212_aCh2_bWrongParameters OR
	DiagsRetain.DG_REM10_PO1212_aCh3_bOpenSensor OR
	DiagsRetain.DG_REM10_PO1212_aCh3_bOverRange OR
	DiagsRetain.DG_REM10_PO1212_aCh3_bSensorShortCircuit OR
	DiagsRetain.DG_REM10_PO1212_aCh3_bWrongParameters OR
	DiagsRetain.DG_REM10_PO1212_aCh4_bOpenSensor OR
	DiagsRetain.DG_REM10_PO1212_aCh4_bOverRange OR
	DiagsRetain.DG_REM10_PO1212_aCh4_bSensorShortCircuit OR
	DiagsRetain.DG_REM10_PO1212_aCh4_bWrongParameters OR
	DiagsRetain.DG_REM10_PO1212_aCh5_bOpenSensor OR
	DiagsRetain.DG_REM10_PO1212_aCh5_bOverRange OR
	DiagsRetain.DG_REM10_PO1212_aCh5_bSensorShortCircuit OR
	DiagsRetain.DG_REM10_PO1212_aCh5_bWrongParameters OR
	DiagsRetain.DG_REM10_PO1212_aCh6_bOpenSensor OR
	DiagsRetain.DG_REM10_PO1212_aCh6_bOverRange OR
	DiagsRetain.DG_REM10_PO1212_aCh6_bSensorShortCircuit OR
	DiagsRetain.DG_REM10_PO1212_aCh6_bWrongParameters OR
	DiagsRetain.DG_REM10_PO1212_aCh7_bOpenSensor OR
	DiagsRetain.DG_REM10_PO1212_aCh7_bOverRange OR
	DiagsRetain.DG_REM10_PO1212_aCh7_bSensorShortCircuit OR
	DiagsRetain.DG_REM10_PO1212_aCh7_bWrongParameters THEN
		bDiag_Error_PO1212_REM10:= TRUE;
	ELSE
		bDiag_Error_PO1212_REM10:= FALSE;	
	END_IF		
	
	IF		
	//PO2132
	DiagsRetain.DG_REM10_PO2132_bNoParametrizedModule OR
	DiagsRetain.DG_REM10_PO2132_bPowerSupplyFail OR
	DiagsRetain.DG_REM10_PO2132_aCh0_bOpenSensor OR
	DiagsRetain.DG_REM10_PO2132_aCh0_bWrongParameters OR
	DiagsRetain.DG_REM10_PO2132_aCh1_bOpenSensor OR
	DiagsRetain.DG_REM10_PO2132_aCh1_bWrongParameters OR
	DiagsRetain.DG_REM10_PO2132_aCh2_bOpenSensor OR
	DiagsRetain.DG_REM10_PO2132_aCh2_bWrongParameters OR
	DiagsRetain.DG_REM10_PO2132_aCh3_bOpenSensor OR
	DiagsRetain.DG_REM10_PO2132_aCh3_bWrongParameters THEN
		bDiag_Error_PO2132_REM10:= TRUE;
	ELSE
		bDiag_Error_PO2132_REM10:= FALSE;	
	END_IF		
	
	IF		
	//PO9100
	DiagsRetain.DG_REM10_PO9100_bReserved00 THEN
			bDiag_Error_PO9100_REM10:= TRUE;
	ELSE
		bDiag_Error_PO9100_REM10:= FALSE;	
	END_IF	
	
	IF		
	//PO1000
	DiagsRetain.DG_REM04_PO1000_bHardwareFailure OR
	DiagsRetain.DG_REM04_PO1000_bPowerSupplyFail THEN
		bDiag_Error_PO1000_REM04:= TRUE;
	ELSE
		bDiag_Error_PO1000_REM04:= FALSE;	
	END_IF	
	
	
	IF 
		bDiag_Error_NX3030 OR
		bDiag_Error_NX4010 OR
		bDiag_Error_NX5001_1 OR
		bDiag_Error_NX5001_2 OR
		bDiag_Error_NX5001_3 OR
		bDiag_Error_NX5000_1 OR
		bDiag_Error_NX5000_2 OR
		bDiag_Error_NX5000_3 OR
		bDiag_Error_MODBUS_Master_1 OR
		bDiag_Error_MODBUS_Slave_1 OR
		bDiag_Error_MODBUS_Client_2 OR
		bDiag_Error_MODBUS_Server_2 OR
		bDiag_Error_MODBUS_Client_3 OR
		bDiag_Error_MODBUS_Server_3 OR
		bDiag_Error_MODBUS_Client_4 OR
		bDiag_Error_MODBUS_Server_4 OR		
		bDiag_Error_PO1000_REM05 OR
		bDiag_Error_PO2020_REM05 OR
		bDiag_Error_PO9100_REM05 OR
		bDiag_Error_PO1212_REM10 OR
		bDiag_Error_PO2132_REM10 OR
		bDiag_Error_PO9100_REM10 OR
		bDiag_Error_PO1000_REM04 THEN
		PersistentVars.bActiveDiagPlcA:= TRUE;
	ELSE
		PersistentVars.bActiveDiagPlcA:= FALSE;

	END_IF
END_IF

// Se este for o PLCB e ele está no estado ativo...
IF DG_NX4010.tRedundancy.RedDgnLoc.sGeneral_Diag.eRedState = REDUNDANCY_STATE.ACTIVE AND 
   DG_NX4010.tRedundancy.RedDgnLoc.sGeneral_Diag.ePLC_ID = CLUCONF_ID.PLC_B THEN
	IF 		
	// NX3030
		DiagsRetain.DG_NX3030_tSummarized_bAbsentModules OR
		DiagsRetain.DG_NX3030_tSummarized_bAbsentRacks OR
		DiagsRetain.DG_NX3030_tSummarized_bCOM1ConfigError OR
		DiagsRetain.DG_NX3030_tSummarized_bCOM2ConfigError OR
		DiagsRetain.DG_NX3030_tSummarized_bConfigMismatch OR
		DiagsRetain.DG_NX3030_tSummarized_bDuplicatedRacks OR
		DiagsRetain.DG_NX3030_tSummarized_bDuplicatedSlots OR
		DiagsRetain.DG_NX3030_tSummarized_bHardwareFailure OR
		DiagsRetain.DG_NX3030_tSummarized_bInvalidDateTime OR
		DiagsRetain.DG_NX3030_tSummarized_bInvalidRacks OR
		DiagsRetain.DG_NX3030_tSummarized_bMemoryCardError OR
		DiagsRetain.DG_NX3030_tSummarized_bModuleFatalError OR
		DiagsRetain.DG_NX3030_tSummarized_bModuleParameterError OR
		DiagsRetain.DG_NX3030_tSummarized_bModulesWithDiagnostic OR
		DiagsRetain.DG_NX3030_tSummarized_bNET1ConfigError OR
		DiagsRetain.DG_NX3030_tSummarized_bNET2ConfigError OR
		DiagsRetain.DG_NX3030_tSummarized_bNonDeclaredModules OR
		DiagsRetain.DG_NX3030_tSummarized_bNonDeclaredRacks OR
		DiagsRetain.DG_NX3030_tSummarized_bOTDSwitchError OR
		DiagsRetain.DG_NX3030_tSummarized_bRuntimeReset OR
		DiagsRetain.DG_NX3030_tSummarized_bSoftwareException OR
		DiagsRetain.DG_NX3030_tSummarized_bSwappedModules OR
		DiagsRetain.DG_NX3030_tSummarized_bWHSBBusError OR
		DiagsRetain.DG_NX3030_tDetailed_MemoryCard_byMounted OR
		DiagsRetain.DG_NX3030_tDetailed_Ethernet_NET1_bLinkDown OR
		DiagsRetain.DG_NX3030_tDetailed_Ethernet_NET2_bLinkDown OR 
		DiagsRetain.DG_NX3030_tDetailed_Application_byCPUState OR
		DiagsRetain.DG_NX3030_tDetailed_ApplicationInfo_dwApplicationCRC OR
		DiagsRetain.DG_NX3030_tDetailed_Ethernet_NET1_abyMAC_0 OR
		DiagsRetain.DG_NX3030_tDetailed_Ethernet_NET1_abyMAC_1 OR
		DiagsRetain.DG_NX3030_tDetailed_Ethernet_NET1_abyMAC_2 OR
		DiagsRetain.DG_NX3030_tDetailed_Ethernet_NET1_abyMAC_3 OR
		DiagsRetain.DG_NX3030_tDetailed_Ethernet_NET1_abyMAC_4 OR
		DiagsRetain.DG_NX3030_tDetailed_Ethernet_NET1_abyMAC_5 OR
		DiagsRetain.DG_NX3030_tDetailed_Ethernet_NET2_abyMAC_0 OR
		DiagsRetain.DG_NX3030_tDetailed_Ethernet_NET2_abyMAC_1 OR
		DiagsRetain.DG_NX3030_tDetailed_Ethernet_NET2_abyMAC_2 OR
		DiagsRetain.DG_NX3030_tDetailed_Ethernet_NET2_abyMAC_3 OR
		DiagsRetain.DG_NX3030_tDetailed_Ethernet_NET2_abyMAC_4 OR
		DiagsRetain.DG_NX3030_tDetailed_Ethernet_NET2_abyMAC_5 OR
		DiagsRetain.DG_NX3030_tDetailed_Ethernet_NETx_abyIP_0 OR
		DiagsRetain.DG_NX3030_tDetailed_Ethernet_NETx_abyIP_1 OR
		DiagsRetain.DG_NX3030_tDetailed_Ethernet_NETx_abyIP_2 OR
		DiagsRetain.DG_NX3030_tDetailed_Ethernet_NETx_abyIP_3 OR
		DiagsRetain.DG_NX3030_tDetailed_Ethernet_NETx_abyMask_0 OR
		DiagsRetain.DG_NX3030_tDetailed_Ethernet_NETx_abyMask_1 OR
		DiagsRetain.DG_NX3030_tDetailed_Ethernet_NETx_abyMask_2 OR
		DiagsRetain.DG_NX3030_tDetailed_Ethernet_NETx_abyMask_3 OR
		DiagsRetain.DG_NX3030_tDetailed_Ethernet_NETx_abyGateway_0 OR
		DiagsRetain.DG_NX3030_tDetailed_Ethernet_NETx_abyGateway_1 OR
		DiagsRetain.DG_NX3030_tDetailed_Ethernet_NETx_abyGateway_2 OR
		DiagsRetain.DG_NX3030_tDetailed_Ethernet_NETx_abyGateway_3 OR
		DiagsRetain.DG_NX3030_tDetailed_SNTP_bServiceEnabled OR
		DiagsRetain.DG_NX3030_tDetailed_Target_abyAuxprocVersion OR
		DiagsRetain.DG_NX3030_tDetailed_Target_abyBootloaderVersion OR
		DiagsRetain.DG_NX3030_tDetailed_Target_abyCPUVersion OR
		DiagsRetain.DG_NX3030_tDetailed_Target_dwCPUModel OR
		DiagsRetain.DG_NX3030_tDetailed_Thermometer_diTemperature THEN
    bDiag_Error_NX3030:= TRUE;
	ELSE
		bDiag_Error_NX3030:= FALSE;	
	END_IF
	
	IF	
	// NX4010
		DiagsRetain.DG_NX4010_tGeneral_bActiveDiagnostics OR
		DiagsRetain.DG_NX4010_tGeneral_bBusCommunicationError OR
		DiagsRetain.DG_NX4010_tGeneral_bConfigMismatch OR
		DiagsRetain.DG_NX4010_tGeneral_bFatalError OR
		DiagsRetain.DG_NX4010_tGeneral_bNET1LinkDown OR
		DiagsRetain.DG_NX4010_tGeneral_bNET2LinkDown OR
		DiagsRetain.DG_NX4010_tGeneral_bOTDSwitchError OR
		DiagsRetain.DG_NX4010_tGeneral_bWatchdogError OR
		DiagsRetain.DG_NX4010_tRedundancy_RedDgnLoc_sGeneral_Diag_bApplicationIncompatible OR
		DiagsRetain.DG_NX4010_tRedundancy_RedDgnLoc_sGeneral_Diag_bApplicationProjectDiff OR
		DiagsRetain.DG_NX4010_tRedundancy_RedDgnLoc_sGeneral_Diag_bConfigError OR
		DiagsRetain.DG_NX4010_tRedundancy_RedDgnLoc_sGeneral_Diag_bExchangeSync OR
		DiagsRetain.DG_NX4010_tRedundancy_RedDgnLoc_sGeneral_Diag_bFailedPBUS1A OR
		DiagsRetain.DG_NX4010_tRedundancy_RedDgnLoc_sGeneral_Diag_bFailedPBUS1B OR
		DiagsRetain.DG_NX4010_tRedundancy_RedDgnLoc_sGeneral_Diag_bFailedPBUS2A OR
		DiagsRetain.DG_NX4010_tRedundancy_RedDgnLoc_sGeneral_Diag_bFailedPBUS2B OR
		DiagsRetain.DG_NX4010_tRedundancy_RedDgnLoc_sGeneral_Diag_bFailedRED OR
		DiagsRetain.DG_NX4010_tRedundancy_RedDgnLoc_sGeneral_Diag_bFailureProfibus_1 OR
		DiagsRetain.DG_NX4010_tRedundancy_RedDgnLoc_sGeneral_Diag_bFailureProfibus_2 OR
		DiagsRetain.DG_NX4010_tRedundancy_RedDgnLoc_sGeneral_Diag_bIncompatibleFirmware OR
		DiagsRetain.DG_NX4010_tRedundancy_RedDgnLoc_sGeneral_Diag_bProfibusVitalFailureAll OR
		DiagsRetain.DG_NX4010_tRedundancy_RedDgnLoc_sGeneral_Diag_bProfibusVitalFailureAny OR
		DiagsRetain.DG_NX4010_tRedundancy_RedDgnLoc_sGeneral_Diag_bProjectArchiveDiff OR
		DiagsRetain.DG_NX4010_tRedundancy_RedDgnLoc_sGeneral_Diag_bProjectSyncDisable OR
		DiagsRetain.DG_NX4010_tRedundancy_RedDgnLoc_sGeneral_Diag_bRedDataSync OR
		DiagsRetain.DG_NX4010_tRedundancy_RedDgnLoc_sGeneral_Diag_bRedForceSync OR
		DiagsRetain.DG_NX4010_tRedundancy_RedDgnLoc_sGeneral_Diag_bRedPanelTestMode OR
		DiagsRetain.DG_NX4010_tRedundancy_RedDgnLoc_sGeneral_Diag_bTemporaryBufferTooSmall OR
		DiagsRetain.DG_NX4010_tRedundancy_RedDgnLoc_sGeneral_Diag_bTooManyRedAreas OR
		DiagsRetain.DG_NX4010_tRedundancy_RedDgnLoc_sGeneral_Diag_dwArchiveCRC OR  // Demanda 19831
		DiagsRetain.DG_NX4010_tRedundancy_RedDgnLoc_sGeneral_Diag_dwApplicationCRC THEN
    	bDiag_Error_NX4010:= TRUE;
	ELSE
		bDiag_Error_NX4010:= FALSE;	
	END_IF
	
	IF		
	// NX5001_1
		DiagsRetain.DG_NX5001_1_tGeneral_bActiveDiagnostics OR
		DiagsRetain.DG_NX5001_1_tGeneral_bBusCommunicationError OR
		DiagsRetain.DG_NX5001_1_tGeneral_bConfigMismatch OR
		DiagsRetain.DG_NX5001_1_tGeneral_bFatalError OR
		DiagsRetain.DG_NX5001_1_tGeneral_bNX5001NoCfg OR
		DiagsRetain.DG_NX5001_1_tGeneral_bOTDSwitchError OR
		DiagsRetain.DG_NX5001_1_tGeneral_bPbusCommFail OR
		DiagsRetain.DG_NX5001_1_tGeneral_bSlaveNotConfigured OR
		DiagsRetain.DG_NX5001_1_tGeneral_bSlaveNotPresent OR
		DiagsRetain.DG_NX5001_1_tGeneral_bSlaveWithDiagnostic OR
		DiagsRetain.DG_NX5001_1_tGeneral_bStsEnableInterface OR
	//	DiagsRetain.DG_NX5001_1_tGeneral_bStsMstRedundEnable OR   Demanda 17571
		DiagsRetain.DG_NX5001_1_tGeneral_bWatchdogError THEN
    	bDiag_Error_NX5001_1:= TRUE;
	ELSE
		bDiag_Error_NX5001_1:= FALSE;	
	END_IF
	
